C09104=1059.503,108.760,421.956,171.884,30.619,155.688
C09105=1059.497,108.511,421.976,171.883,30.616,155.687
C09106=1059.490,108.261,421.996,171.881,30.614,155.687
C09107=1059.484,108.012,422.014,171.879,30.611,155.687
C09108=1059.478,107.763,422.034,171.878,30.609,155.686
C09109=1059.472,107.514,422.053,171.876,30.606,155.686
C09110=1059.466,107.264,422.073,171.875,30.603,155.685
C09111=1059.460,107.015,422.093,171.873,30.601,155.685
C09112=1059.455,106.766,422.112,171.871,30.598,155.685
C09113=1059.448,106.517,422.131,171.870,30.596,155.684
C09114=1059.442,106.268,422.150,171.868,30.593,155.684
C09115=1059.437,106.019,422.170,171.867,30.591,155.683
C09116=1059.431,105.769,422.189,171.865,30.588,155.683
C09117=1059.424,105.521,422.208,171.863,30.585,155.683
C09118=1059.419,105.271,422.228,171.862,30.583,155.682
C09119=1059.413,105.022,422.247,171.861,30.580,155.682
C09120=1059.407,104.773,422.267,171.859,30.577,155.681
C09121=1059.401,104.524,422.286,171.857,30.575,155.681
C09122=1059.395,104.274,422.305,171.855,30.573,155.681
C09123=1059.389,104.025,422.324,171.854,30.570,155.680
C09124=1059.383,103.776,422.344,171.853,30.567,155.680
C09125=1059.377,103.527,422.363,171.851,30.565,155.679
C09126=1059.371,103.278,422.382,171.849,30.562,155.679
C09127=1059.365,103.028,422.401,171.847,30.559,155.679
C09128=1059.359,102.779,422.421,171.846,30.557,155.678
C09129=1059.354,102.531,422.440,171.845,30.554,155.678
C09130=1059.348,102.281,422.459,171.843,30.551,155.677
C09131=1059.342,102.032,422.478,171.841,30.549,155.677
C09132=1059.336,101.783,422.497,171.840,30.547,155.677
C09133=1059.330,101.534,422.517,171.839,30.544,155.676
C09134=1059.325,101.284,422.536,171.837,30.541,155.676
C09135=1059.318,101.035,422.555,171.835,30.539,155.675
C09136=1059.313,100.786,422.574,171.833,30.536,155.675
C09137=1059.306,100.537,422.593,171.832,30.533,155.675
C09138=1059.300,100.287,422.612,171.831,30.531,155.674
C09139=1059.295,100.038,422.631,171.829,30.529,155.674
C09140=1059.288,99.789,422.650,171.827,30.526,155.674
C09141=1059.283,99.539,422.669,171.825,30.523,155.673
C09142=1059.276,99.291,422.688,171.824,30.521,155.673
C09143=1059.270,99.041,422.708,171.823,30.518,155.672
C09144=1059.264,98.792,422.726,171.821,30.516,155.672
C09145=1059.258,98.543,422.746,171.819,30.513,155.672
C09146=1059.252,98.294,422.764,171.818,30.511,155.671
C09147=1059.247,98.045,422.783,171.817,30.508,155.671
C09148=1059.240,97.796,422.802,171.815,30.505,155.670
C09149=1059.234,97.546,422.821,171.813,30.503,155.670
C09150=1059.228,97.297,422.840,171.811,30.501,155.670
C09151=1059.222,97.048,422.859,171.810,30.498,155.669
C09152=1059.216,96.799,422.878,171.809,30.495,155.669
C09153=1059.210,96.549,422.897,171.807,30.493,155.668
C09154=1059.204,96.300,422.915,171.805,30.491,155.668
C09155=1059.198,96.051,422.935,171.804,30.488,155.668
C09156=1059.192,95.802,422.953,171.802,30.485,155.667
C09157=1059.187,95.553,422.972,171.801,30.483,155.667
C09158=1059.180,95.304,422.991,171.799,30.480,155.666
C09159=1059.175,95.054,423.010,171.797,30.477,155.666
C09160=1059.168,94.805,423.029,171.796,30.475,155.666
C09161=1059.162,94.520,423.050,171.795,30.472,155.665
C09162=1059.155,94.235,423.072,171.793,30.469,155.665
C09163=1059.148,93.951,423.093,171.791,30.466,155.664
C09164=1059.142,93.666,423.115,171.789,30.463,155.664
C09165=1059.135,93.417,423.133,171.788,30.461,155.663
C09166=1059.129,93.168,423.153,171.786,30.458,155.663
C09167=1059.123,92.919,423.171,171.784,30.455,155.663
C09168=1059.118,92.669,423.190,171.782,30.453,155.662
C09169=1059.111,92.420,423.208,171.781,30.451,155.662
C09170=1059.106,92.171,423.227,171.780,30.448,155.662
C09171=1059.100,91.922,423.246,171.778,30.445,155.661
C09172=1059.094,91.672,423.265,171.776,30.442,155.661
C09173=1059.088,91.423,423.284,171.775,30.440,155.660
C09174=1059.083,91.174,423.302,171.774,30.437,155.660
C09175=1059.076,90.925,423.321,171.772,30.435,155.660
C09176=1059.071,90.675,423.340,171.770,30.432,155.659
C09177=1059.064,90.426,423.358,171.769,30.430,155.659
C09178=1059.058,90.177,423.377,171.767,30.427,155.658
C09179=1059.052,89.927,423.395,171.766,30.424,155.658
C09180=1059.046,89.679,423.413,171.764,30.422,155.658
C09181=1059.040,89.429,423.433,171.763,30.420,155.657
C09182=1059.034,89.180,423.451,171.761,30.417,155.657
C09183=1059.028,88.931,423.469,171.759,30.415,155.656
C09184=1059.021,88.681,423.488,171.758,30.412,155.656
C09185=1059.015,88.432,423.507,171.756,30.410,155.656
C09186=1059.010,88.183,423.525,171.755,30.407,155.655
C09187=1059.004,87.934,423.543,171.753,30.405,155.655
C09188=1058.997,87.685,423.562,171.752,30.402,155.655
C09189=1058.991,87.435,423.580,171.750,30.400,155.654
C09190=1058.985,87.185,423.599,171.749,30.397,155.654
C09191=1058.979,86.937,423.617,171.747,30.395,155.653
C09192=1058.973,86.687,423.635,171.745,30.392,155.653
C09193=1058.967,86.438,423.654,171.744,30.389,155.653
C09194=1058.961,86.189,423.673,171.743,30.387,155.652
C09195=1058.956,85.940,423.691,171.741,30.384,155.652
C09196=1058.949,85.691,423.709,171.739,30.382,155.652
C09197=1058.943,85.442,423.728,171.738,30.379,155.651
C09198=1058.937,85.192,423.746,171.737,30.377,155.651
C09199=1058.931,84.943,423.764,171.735,30.374,155.650
C09200=1058.926,84.693,423.783,171.733,30.372,155.650
C09201=1058.919,84.444,423.801,171.731,30.369,155.650
C09202=1058.913,84.195,423.820,171.731,30.367,155.649
C09203=1058.907,83.946,423.838,171.729,30.364,155.649
C09204=1058.901,83.697,423.856,171.727,30.361,155.648
C09205=1058.895,83.447,423.875,171.725,30.359,155.648
C09206=1058.890,83.198,423.893,171.725,30.357,155.648
C09207=1058.883,82.949,423.911,171.723,30.354,155.647
C09208=1058.877,82.700,423.930,171.721,30.351,155.647
C09209=1058.871,82.450,423.948,171.719,30.349,155.646
C09210=1058.865,82.201,423.966,171.719,30.347,155.646
C09211=1058.860,81.951,423.984,171.717,30.344,155.646
C09212=1058.853,81.702,424.003,171.715,30.341,155.645
C09213=1058.848,81.453,424.021,171.713,30.338,155.645
C09214=1058.841,81.204,424.039,171.712,30.336,155.644
C09215=1058.835,80.954,424.057,171.711,30.334,155.644
C09216=1058.829,80.706,424.076,171.709,30.331,155.644
C09217=1058.823,80.456,424.093,171.707,30.328,155.643
C09218=1058.818,80.207,424.113,171.706,30.326,155.643
C09219=1058.812,79.958,424.130,171.705,30.323,155.643
C09220=1058.806,79.708,424.148,171.703,30.321,155.642
C09221=1058.800,79.460,424.166,171.701,30.318,155.642
C09222=1058.794,79.210,424.184,171.700,30.316,155.641
C09223=1058.788,78.961,424.203,171.699,30.313,155.641
C09224=1058.782,78.712,424.221,171.697,30.310,155.641
C09225=1058.773,78.312,424.250,171.694,30.306,155.640
C09226=1058.763,77.912,424.279,171.692,30.302,155.639
C09227=1058.753,77.512,424.308,171.690,30.298,155.639
C09228=1058.743,77.114,424.336,171.687,30.294,155.638
C09229=1058.737,76.864,424.354,171.685,30.292,155.638
C09230=1058.731,76.615,424.373,171.684,30.289,155.637
C09231=1058.725,76.366,424.391,171.683,30.287,155.637
C09232=1058.719,76.116,424.409,171.681,30.284,155.637
C09233=1058.713,75.867,424.427,171.679,30.282,155.636
C09234=1058.707,75.618,424.445,171.678,30.279,155.636
C09235=1058.701,75.368,424.463,171.677,30.277,155.635
C09236=1058.696,75.119,424.480,171.675,30.275,155.635
C09237=1058.689,74.870,424.498,171.673,30.272,155.635
C09238=1058.682,74.620,424.516,171.672,30.269,155.634
C09239=1058.677,74.371,424.534,171.671,30.267,155.634
C09240=1058.671,74.122,424.552,171.669,30.265,155.634
C09241=1058.665,73.873,424.570,171.667,30.262,155.633
C09242=1058.659,73.623,424.588,171.665,30.259,155.633
C09243=1058.653,73.374,424.606,171.665,30.257,155.632
C09244=1058.647,73.125,424.623,171.663,30.254,155.632
C09245=1058.641,72.876,424.642,171.661,30.252,155.632
C09246=1058.635,72.627,424.659,171.660,30.249,155.631
C09247=1058.628,72.377,424.677,171.659,30.246,155.631
C09248=1058.623,72.128,424.695,171.657,30.244,155.631
C09249=1058.617,71.878,424.713,171.655,30.242,155.630
C09250=1058.611,71.629,424.730,171.654,30.239,155.630
C09251=1058.605,71.380,424.749,171.652,30.237,155.630
C09252=1058.599,71.130,424.767,171.651,30.234,155.629
C09253=1058.592,70.882,424.784,171.649,30.232,155.629
C09254=1058.586,70.632,424.802,171.648,30.229,155.628
C09255=1058.581,70.383,424.819,171.646,30.227,155.628
C09256=1058.575,70.133,424.837,171.645,30.224,155.628
C09257=1058.569,69.884,424.855,171.643,30.221,155.627
C09258=1058.563,69.634,424.873,171.642,30.219,155.627
C09259=1058.557,69.386,424.890,171.640,30.217,155.626
C09260=1058.551,69.136,424.908,171.639,30.214,155.626
C09261=1058.541,68.752,424.935,171.636,30.210,155.625
C09262=1058.532,68.368,424.962,171.634,30.207,155.625
C09263=1058.522,67.985,424.989,171.632,30.203,155.624
C09264=1058.513,67.601,425.016,171.629,30.198,155.624
C09265=1058.508,67.352,425.034,171.628,30.196,155.623
C09266=1058.501,67.102,425.051,171.626,30.194,155.623
C09267=1058.495,66.852,425.069,171.625,30.191,155.623
C09268=1058.489,66.603,425.087,171.623,30.189,155.622
C09269=1058.483,66.354,425.104,171.622,30.186,155.622
C09270=1058.477,66.105,425.122,171.620,30.184,155.622
C09271=1058.471,65.855,425.140,171.619,30.181,155.621
C09272=1058.465,65.606,425.157,171.617,30.179,155.621
C09273=1058.459,65.357,425.175,171.616,30.176,155.620
C09274=1058.453,65.108,425.192,171.614,30.174,155.620
C09275=1058.447,64.859,425.209,171.613,30.171,155.620
C09276=1058.441,64.609,425.227,171.612,30.169,155.619
C09277=1058.435,64.360,425.245,171.610,30.166,155.619
C09278=1058.429,64.110,425.261,171.608,30.164,155.619
C09279=1058.422,63.860,425.279,171.607,30.161,155.618
C09280=1058.416,63.612,425.296,171.606,30.159,155.618
C09281=1058.409,63.362,425.313,171.604,30.157,155.617
C09282=1058.404,63.113,425.331,171.602,30.154,155.617
C09283=1058.397,62.864,425.348,171.600,30.152,155.617
C09284=1058.391,62.615,425.366,171.599,30.149,155.616
C09285=1058.384,62.330,425.385,171.597,30.146,155.616
C09286=1058.377,62.044,425.406,171.595,30.144,155.616
C09287=1058.370,61.760,425.425,171.594,30.141,155.615
C09288=1058.363,61.475,425.444,171.592,30.138,155.615
C09289=1058.357,61.226,425.462,171.591,30.136,155.614
C09290=1058.350,60.976,425.478,171.589,30.133,155.614
C09291=1058.345,60.727,425.496,171.588,30.131,155.614
C09292=1058.338,60.478,425.513,171.587,30.129,155.613
C09293=1058.332,60.229,425.530,171.585,30.126,155.613
C09294=1058.326,59.979,425.548,171.583,30.124,155.613
C09295=1058.320,59.730,425.565,171.581,30.121,155.612
C09296=1058.314,59.480,425.582,171.581,30.119,155.612
C09297=1058.307,59.231,425.599,171.579,30.116,155.612
C09298=1058.301,58.981,425.616,171.577,30.114,155.611
C09299=1058.295,58.732,425.634,171.575,30.112,155.611
C09300=1058.289,58.484,425.651,171.575,30.109,155.610
C09301=1058.283,58.233,425.668,171.573,30.106,155.610
C09302=1058.277,57.985,425.685,171.571,30.104,155.610
C09303=1058.270,57.735,425.702,171.569,30.101,155.609
C09304=1058.265,57.485,425.719,171.569,30.099,155.609
C09305=1058.258,57.236,425.736,171.567,30.097,155.609
C09306=1058.253,56.987,425.754,171.565,30.094,155.608
C09307=1058.247,56.738,425.770,171.563,30.092,155.608
C09308=1058.240,56.488,425.787,171.562,30.089,155.608
C09309=1058.234,56.239,425.805,171.561,30.087,155.607
C09310=1058.228,55.990,425.821,171.559,30.084,155.607
C09311=1058.221,55.740,425.839,171.557,30.082,155.606
C09312=1058.216,55.491,425.856,171.556,30.080,155.606
C09313=1058.209,55.241,425.873,171.555,30.077,155.606
C09314=1058.203,54.993,425.890,171.553,30.075,155.605
C09315=1058.198,54.743,425.907,171.551,30.072,155.605
C09316=1058.191,54.493,425.924,171.550,30.070,155.605
C09317=1058.185,54.244,425.942,171.549,30.067,155.604
C09318=1058.180,53.995,425.958,171.547,30.065,155.604
C09319=1058.173,53.746,425.975,171.545,30.063,155.604
C09320=1058.167,53.496,425.992,171.544,30.060,155.603
C09321=1058.161,53.247,426.009,171.543,30.057,155.603
C09322=1058.155,52.997,426.026,171.541,30.055,155.603
C09323=1058.149,52.748,426.043,171.539,30.052,155.602
C09324=1058.143,52.499,426.059,171.538,30.050,155.602
C09325=1058.136,52.249,426.077,171.537,30.048,155.601
C09326=1058.131,52.000,426.094,171.535,30.045,155.601
C09327=1058.125,51.751,426.111,171.533,30.043,155.601
C09328=1058.118,51.501,426.127,171.532,30.040,155.600
C09329=1058.113,51.252,426.145,171.531,30.037,155.600
C09330=1058.107,51.003,426.161,171.529,30.035,155.600
C09331=1058.101,50.754,426.178,171.527,30.033,155.599
C09332=1058.094,50.504,426.195,171.526,30.030,155.599
C09333=1058.089,50.255,426.212,171.525,30.028,155.599
C09334=1058.083,50.005,426.228,171.523,30.025,155.598
C09335=1058.076,49.757,426.245,171.522,30.023,155.598
C09336=1058.070,49.506,426.263,171.520,30.020,155.597
C09337=1058.065,49.257,426.279,171.519,30.018,155.597
C09338=1058.058,49.008,426.296,171.517,30.016,155.597
C09339=1058.053,48.759,426.313,171.516,30.013,155.596
C09340=1058.046,48.509,426.330,171.514,30.010,155.596
C09341=1058.040,48.260,426.346,171.513,30.008,155.596
C09342=1058.035,48.010,426.363,171.511,30.005,155.595
C09343=1058.029,47.761,426.380,171.510,30.003,155.595
C09344=1058.022,47.511,426.397,171.508,30.001,155.595
C09345=1058.016,47.263,426.414,171.507,29.998,155.594
C09346=1058.011,47.013,426.431,171.505,29.995,155.594
C09347=1058.005,46.764,426.447,171.504,29.993,155.593
C09348=1057.999,46.515,426.464,171.502,29.991,155.593
C09349=1057.992,46.229,426.483,171.501,29.988,155.593
C09350=1057.985,45.943,426.502,171.499,29.985,155.592
C09351=1057.978,45.659,426.521,171.497,29.982,155.592
C09352=1057.971,45.373,426.541,171.495,29.979,155.591
C09353=1057.965,45.124,426.557,171.494,29.977,155.591
C09354=1057.959,44.875,426.574,171.492,29.974,155.591
C09355=1057.953,44.626,426.590,171.491,29.972,155.590
C09356=1057.948,44.376,426.607,171.489,29.969,155.590
C09357=1057.942,44.127,426.623,171.488,29.967,155.590
C09358=1057.935,43.877,426.641,171.487,29.964,155.589
C09359=1057.929,43.628,426.657,171.485,29.962,155.589
C09360=1057.924,43.378,426.674,171.483,29.959,155.588
C09361=1057.918,43.129,426.690,171.482,29.957,155.588
C09362=1057.912,42.880,426.706,171.481,29.954,155.588
C09363=1057.905,42.630,426.724,171.479,29.952,155.587
C09364=1057.899,42.381,426.740,171.477,29.950,155.587
C09365=1057.893,42.132,426.756,171.476,29.947,155.587
C09366=1057.887,41.882,426.772,171.475,29.945,155.586
C09367=1057.881,41.633,426.789,171.473,29.943,155.586
C09368=1057.875,41.384,426.806,171.471,29.940,155.586
C09369=1057.869,41.134,426.822,171.470,29.937,155.585
C09370=1057.863,40.885,426.838,171.468,29.935,155.585
C09371=1057.857,40.635,426.855,171.467,29.932,155.585
C09372=1057.851,40.386,426.871,171.465,29.930,155.584
C09373=1057.845,40.137,426.887,171.464,29.928,155.584
C09374=1057.839,39.887,426.903,171.462,29.925,155.584
C09375=1057.832,39.637,426.920,171.461,29.923,155.583
C09376=1057.826,39.389,426.937,171.459,29.921,155.583
C09377=1057.820,39.139,426.953,171.458,29.918,155.583
C09378=1057.814,38.890,426.970,171.456,29.916,155.582
C09379=1057.808,38.641,426.986,171.455,29.913,155.582
C09380=1057.802,38.391,427.002,171.453,29.911,155.581
C09381=1057.796,38.142,427.018,171.452,29.908,155.581
C09382=1057.790,37.893,427.035,171.450,29.906,155.581
C09383=1057.784,37.642,427.051,171.449,29.904,155.580
C09384=1057.778,37.393,427.067,171.447,29.901,155.580
C09385=1057.772,37.144,427.084,171.446,29.899,155.580
C09386=1057.766,36.894,427.100,171.444,29.897,155.579
C09387=1057.759,36.645,427.116,171.443,29.894,155.579
C09388=1057.753,36.396,427.132,171.441,29.892,155.579
C09389=1057.747,36.147,427.148,171.440,29.889,155.578
C09390=1057.741,35.897,427.165,171.438,29.887,155.578
C09391=1057.735,35.647,427.181,171.437,29.884,155.578
C09392=1057.728,35.398,427.197,171.435,29.882,155.577
C09393=1057.722,35.149,427.213,171.434,29.879,155.577
C09394=1057.716,34.900,427.229,171.432,29.877,155.577
C09395=1057.710,34.650,427.245,171.431,29.875,155.576
C09396=1057.704,34.401,427.262,171.429,29.873,155.576
C09397=1057.698,34.152,427.278,171.428,29.870,155.576
C09398=1057.692,33.902,427.293,171.426,29.868,155.575
C09399=1057.686,33.653,427.309,171.424,29.866,155.575
C09400=1057.680,33.402,427.326,171.423,29.863,155.575
C09401=1057.674,33.153,427.342,171.422,29.861,155.574
C09402=1057.667,32.904,427.358,171.420,29.858,155.574
C09403=1057.661,32.655,427.374,171.418,29.856,155.574
C09404=1057.655,32.405,427.390,171.417,29.853,155.573
C09405=1057.649,32.156,427.406,171.416,29.851,155.573
C09406=1057.643,31.906,427.422,171.414,29.849,155.573
C09407=1057.637,31.657,427.438,171.412,29.846,155.572
C09408=1057.631,31.408,427.454,171.411,29.844,155.572
C09409=1057.625,31.158,427.470,171.410,29.842,155.572
C09410=1057.619,30.909,427.486,171.408,29.839,155.571
C09411=1057.613,30.660,427.503,171.406,29.837,155.571
C09412=1057.606,30.410,427.518,171.405,29.835,155.571
C09413=1057.599,30.125,427.537,171.404,29.832,155.570
C09414=1057.593,29.840,427.555,171.402,29.829,155.570
C09415=1057.586,29.554,427.573,171.399,29.826,155.569
C09416=1057.579,29.270,427.590,171.398,29.823,155.569
C09417=1057.573,29.020,427.607,171.397,29.821,155.569
C09418=1057.567,28.771,427.623,171.395,29.819,155.568
C09419=1057.561,28.521,427.639,171.393,29.817,155.568
C09420=1057.555,28.272,427.654,171.392,29.814,155.568
C09421=1057.549,28.022,427.670,171.391,29.812,155.567
C09422=1057.542,27.773,427.686,171.389,29.810,155.567
C09423=1057.536,27.523,427.702,171.387,29.807,155.567
C09424=1057.530,27.274,427.718,171.386,29.805,155.566
C09425=1057.524,27.025,427.734,171.385,29.802,155.566
C09426=1057.518,26.775,427.749,171.383,29.800,155.566
C09427=1057.511,26.526,427.765,171.381,29.798,155.565
C09428=1057.505,26.277,427.781,171.380,29.795,155.565
C09429=1057.500,26.027,427.797,171.378,29.793,155.565
C09430=1057.493,25.778,427.812,171.377,29.791,155.564
C09431=1057.487,25.528,427.828,171.375,29.788,155.564
C09432=1057.481,25.279,427.843,171.374,29.786,155.564
C09433=1057.475,25.029,427.860,171.372,29.784,155.564
C09434=1057.468,24.780,427.875,171.370,29.781,155.563
C09435=1057.462,24.530,427.891,171.369,29.779,155.563
C09436=1057.456,24.281,427.907,171.368,29.776,155.562
C09437=1057.450,24.031,427.922,171.366,29.774,155.562
C09438=1057.444,23.782,427.938,171.364,29.772,155.562
C09439=1057.437,23.533,427.954,171.363,29.769,155.561
C09440=1057.432,23.283,427.970,171.362,29.767,155.561
C09441=1057.425,23.034,427.985,171.360,29.765,155.561
C09442=1057.419,22.784,428.001,171.358,29.762,155.560
C09443=1057.413,22.535,428.016,171.356,29.760,155.560
C09444=1057.407,22.285,428.032,171.356,29.758,155.560
C09445=1057.400,22.036,428.048,171.354,29.755,155.559
C09446=1057.395,21.786,428.063,171.352,29.753,155.559
C09447=1057.388,21.537,428.079,171.350,29.751,155.559
C09448=1057.382,21.287,428.094,171.350,29.749,155.559
C09449=1057.376,21.039,428.110,171.348,29.746,155.558
C09450=1057.371,20.789,428.125,171.346,29.744,155.558
C09451=1057.364,20.540,428.141,171.344,29.741,155.558
C09452=1057.358,20.290,428.156,171.343,29.739,155.557
C09453=1057.352,20.041,428.172,171.342,29.737,155.557
C09454=1057.346,19.791,428.188,171.340,29.735,155.557
C09455=1057.339,19.542,428.203,171.338,29.732,155.556
C09456=1057.334,19.292,428.219,171.337,29.730,155.556
C09457=1057.327,19.042,428.234,171.335,29.727,155.556
C09458=1057.321,18.793,428.249,171.334,29.725,155.555
C09459=1057.316,18.544,428.265,171.332,29.723,155.555
C09460=1057.309,18.295,428.280,171.331,29.721,155.555
C09461=1057.303,18.045,428.296,171.329,29.718,155.554
C09462=1057.297,17.795,428.311,171.327,29.716,155.554
C09463=1057.290,17.546,428.326,171.326,29.714,155.554
C09464=1057.285,17.296,428.342,171.325,29.711,155.553
C09465=1057.278,17.047,428.358,171.323,29.709,155.553
C09466=1057.272,16.797,428.373,171.321,29.707,155.553
C09467=1057.266,16.548,428.388,171.319,29.704,155.552
C09468=1057.260,16.299,428.403,171.319,29.702,155.552
C09469=1057.254,16.049,428.419,171.317,29.700,155.552
C09470=1057.248,15.799,428.434,171.315,29.697,155.551
C09471=1057.241,15.550,428.450,171.313,29.695,155.551
C09472=1057.235,15.300,428.465,171.312,29.693,155.551
C09473=1057.230,15.051,428.480,171.311,29.691,155.551
C09474=1057.223,14.802,428.495,171.309,29.688,155.550
C09475=1057.217,14.552,428.511,171.307,29.686,155.550
C09476=1057.211,14.303,428.526,171.306,29.684,155.550
C09477=1057.204,14.020,428.543,171.304,29.681,155.549
C09478=1057.197,13.735,428.560,171.302,29.679,155.549
C09479=1057.190,13.451,428.577,171.301,29.676,155.549
C09480=1057.183,13.168,428.595,171.299,29.674,155.548
C09481=1057.177,12.918,428.610,171.297,29.671,155.548
C09482=1057.170,12.668,428.625,171.295,29.669,155.548
C09483=1057.164,12.419,428.640,171.295,29.667,155.547
C09484=1057.157,12.170,428.656,171.293,29.665,155.547
C09485=1057.151,11.921,428.670,171.291,29.663,155.547
C09486=1057.145,11.671,428.685,171.289,29.660,155.546
C09487=1057.139,11.421,428.701,171.288,29.658,155.546
C09488=1057.133,11.171,428.716,171.286,29.656,155.546
C09489=1057.127,10.922,428.731,171.285,29.654,155.546
C09490=1057.120,10.673,428.746,171.283,29.652,155.545
C09491=1057.114,10.424,428.761,171.282,29.649,155.545
C09492=1057.108,10.174,428.776,171.280,29.647,155.545
C09493=1057.101,9.925,428.791,171.278,29.644,155.544
C09494=1057.095,9.675,428.806,171.277,29.642,155.544
C09495=1057.089,9.425,428.821,171.276,29.640,155.544
C09496=1057.084,9.176,428.836,171.274,29.638,155.543
C09497=1057.077,8.926,428.851,171.272,29.636,155.543
C09498=1057.071,8.677,428.866,171.270,29.634,155.543
C09499=1057.064,8.428,428.881,171.269,29.631,155.543
C09500=1057.058,8.179,428.896,171.268,29.629,155.542
C09501=1057.052,7.929,428.911,171.266,29.627,155.542
C09502=1057.046,7.679,428.926,171.264,29.625,155.542
C09503=1057.039,7.430,428.941,171.263,29.622,155.541
C09504=1057.033,7.181,428.955,171.261,29.620,155.541
C09505=1057.028,6.931,428.971,171.260,29.618,155.541
C09506=1057.021,6.681,428.986,171.258,29.616,155.540
C09507=1057.015,6.431,429.001,171.257,29.613,155.540
C09508=1057.009,6.182,429.015,171.255,29.611,155.540
C09509=1057.003,5.933,429.030,171.253,29.609,155.540
C09510=1056.996,5.683,429.045,171.251,29.607,155.539
C09511=1056.991,5.434,429.060,171.251,29.605,155.539
C09512=1056.984,5.185,429.075,171.249,29.603,155.539
C09513=1056.978,4.935,429.090,171.247,29.600,155.538
C09514=1056.972,4.686,429.104,171.245,29.598,155.538
C09515=1056.966,4.436,429.119,171.244,29.596,155.538
C09516=1056.959,4.187,429.134,171.242,29.593,155.538
C09517=1056.953,3.937,429.149,171.241,29.591,155.537
C09518=1056.948,3.688,429.164,171.239,29.589,155.537
C09519=1056.942,3.437,429.179,171.238,29.587,155.537
C09520=1056.935,3.188,429.194,171.236,29.584,155.536
C09521=1056.930,2.939,429.208,171.234,29.582,155.536
C09522=1056.923,2.689,429.223,171.232,29.580,155.536
C09523=1056.917,2.439,429.238,171.232,29.578,155.535
C09524=1056.911,2.191,429.253,171.230,29.576,155.535
C09525=1056.905,1.941,429.268,171.228,29.574,155.535
C09526=1056.899,1.692,429.282,171.226,29.571,155.535
C09527=1056.893,1.442,429.297,171.225,29.569,155.534
C09528=1056.886,1.192,429.311,171.223,29.566,155.534
C09529=1056.881,0.943,429.326,171.222,29.564,155.534
C09530=1056.874,0.693,429.341,171.220,29.562,155.533
C09531=1056.868,0.444,429.356,171.219,29.560,155.533
C09532=1056.862,0.195,429.370,171.217,29.558,155.533
C09533=1056.856,-0.055,429.385,171.215,29.556,155.533
C09534=1056.850,-0.304,429.399,171.213,29.553,155.532
C09535=1056.844,-0.554,429.414,171.213,29.551,155.532
C09536=1056.838,-0.803,429.429,171.211,29.549,155.532
C09537=1056.832,-1.053,429.444,171.209,29.547,155.531
C09538=1056.825,-1.302,429.459,171.208,29.544,155.531
C09539=1056.820,-1.552,429.472,171.206,29.542,155.531
C09540=1056.814,-1.802,429.487,171.204,29.540,155.530
C09541=1056.807,-2.084,429.504,171.202,29.537,155.530
C09542=1056.801,-2.365,429.520,171.201,29.535,155.530
C09543=1056.794,-2.647,429.537,171.199,29.532,155.529
C09544=1056.786,-2.929,429.553,171.197,29.530,155.529
C09545=1056.780,-3.178,429.568,171.195,29.528,155.529
C09546=1056.774,-3.428,429.582,171.194,29.526,155.529
C09547=1056.768,-3.678,429.597,171.192,29.523,155.528
C09548=1056.762,-3.927,429.612,171.191,29.521,155.528
C09549=1056.756,-4.177,429.626,171.189,29.519,155.528
C09550=1056.750,-4.426,429.640,171.188,29.517,155.527
C09551=1056.743,-4.676,429.655,171.186,29.515,155.527
C09552=1056.737,-4.926,429.669,171.184,29.513,155.527
C09553=1056.731,-5.174,429.683,171.182,29.511,155.527
C09554=1056.724,-5.424,429.698,171.181,29.508,155.526
C09555=1056.719,-5.674,429.712,171.180,29.506,155.526
C09556=1056.712,-5.923,429.727,171.178,29.504,155.526
C09557=1056.706,-6.173,429.740,171.176,29.502,155.526
C09558=1056.700,-6.422,429.755,171.175,29.500,155.525
C09559=1056.693,-6.672,429.770,171.173,29.498,155.525
C09560=1056.687,-6.921,429.783,171.171,29.496,155.525
C09561=1056.681,-7.171,429.798,171.169,29.494,155.525
C09562=1056.675,-7.420,429.812,171.168,29.492,155.524
C09563=1056.669,-7.670,429.827,171.167,29.490,155.524
C09564=1056.663,-7.919,429.840,171.165,29.487,155.524
C09565=1056.656,-8.169,429.855,171.163,29.485,155.523
C09566=1056.651,-8.418,429.870,171.162,29.483,155.523
C09567=1056.644,-8.668,429.883,171.160,29.481,155.523
C09568=1056.638,-8.917,429.898,171.158,29.479,155.523
C09569=1056.632,-9.167,429.912,171.156,29.477,155.522
C09570=1056.625,-9.417,429.926,171.155,29.474,155.522
C09571=1056.619,-9.666,429.940,171.154,29.472,155.522
C09572=1056.614,-9.915,429.955,171.152,29.470,155.521
C09573=1056.607,-10.165,429.969,171.150,29.469,155.521
C09574=1056.601,-10.414,429.983,171.149,29.466,155.521
C09575=1056.595,-10.664,429.997,171.147,29.464,155.521
C09576=1056.589,-10.914,430.011,171.145,29.462,155.520
C09577=1056.582,-11.163,430.026,171.143,29.460,155.520
C09578=1056.577,-11.413,430.039,171.142,29.458,155.520
C09579=1056.570,-11.662,430.054,171.141,29.456,155.520
C09580=1056.564,-11.912,430.068,171.139,29.453,155.519
C09581=1056.558,-12.161,430.083,171.137,29.451,155.519
C09582=1056.552,-12.411,430.096,171.136,29.449,155.519
C09583=1056.545,-12.661,430.110,171.134,29.447,155.519
C09584=1056.540,-12.910,430.125,171.132,29.445,155.518
C09585=1056.533,-13.159,430.138,171.130,29.443,155.518
C09586=1056.527,-13.409,430.153,171.129,29.441,155.518
C09587=1056.522,-13.658,430.167,171.127,29.439,155.518
C09588=1056.515,-13.908,430.180,171.126,29.437,155.517
C09589=1056.509,-14.157,430.195,171.124,29.434,155.517
C09590=1056.503,-14.408,430.209,171.123,29.432,155.517
C09591=1056.497,-14.657,430.222,171.121,29.430,155.516
C09592=1056.491,-14.906,430.237,171.119,29.429,155.516
C09593=1056.485,-15.156,430.251,171.117,29.426,155.516
C09594=1056.479,-15.405,430.265,171.116,29.424,155.516
C09595=1056.472,-15.655,430.279,171.114,29.422,155.515
C09596=1056.466,-15.904,430.293,171.112,29.420,155.515
C09597=1056.459,-16.154,430.306,171.111,29.418,155.515
C09598=1056.454,-16.404,430.320,171.110,29.416,155.515
C09599=1056.447,-16.652,430.334,171.108,29.414,155.514
C09600=1056.441,-16.903,430.348,171.106,29.412,155.514
C09601=1056.435,-17.152,430.362,171.104,29.410,155.514
C09602=1056.428,-17.402,430.375,171.103,29.408,155.514
C09603=1056.422,-17.651,430.390,171.101,29.406,155.514
C09604=1056.416,-17.900,430.403,171.099,29.404,155.513
C09605=1056.409,-18.181,430.419,171.098,29.401,155.513
C09606=1056.402,-18.461,430.434,171.096,29.399,155.513
C09607=1056.395,-18.742,430.450,171.094,29.397,155.512
C09608=1056.389,-19.022,430.466,171.092,29.395,155.512
C09609=1056.382,-19.271,430.479,171.091,29.393,155.512
C09610=1056.376,-19.521,430.492,171.089,29.391,155.512
C09611=1056.370,-19.770,430.507,171.087,29.389,155.511
C09612=1056.364,-20.020,430.520,171.085,29.387,155.511
C09613=1056.358,-20.270,430.535,171.084,29.385,155.511
C09614=1056.351,-20.519,430.548,171.082,29.383,155.511
C09615=1056.345,-20.768,430.561,171.080,29.381,155.510
C09616=1056.339,-21.019,430.575,171.078,29.378,155.510
C09617=1056.333,-21.268,430.589,171.077,29.377,155.510
C09618=1056.326,-21.517,430.603,171.075,29.375,155.510
C09619=1056.320,-21.767,430.617,171.074,29.373,155.509
C09620=1056.314,-22.016,430.630,171.072,29.371,155.509
C09621=1056.308,-22.266,430.644,171.071,29.369,155.509
C09622=1056.302,-22.516,430.658,171.069,29.367,155.509
C09623=1056.295,-22.765,430.671,171.067,29.364,155.509
C09624=1056.290,-23.015,430.685,171.065,29.363,155.508
C09625=1056.283,-23.264,430.698,171.064,29.361,155.508
C09626=1056.277,-23.514,430.712,171.062,29.358,155.508
C09627=1056.271,-23.763,430.725,171.060,29.357,155.508
C09628=1056.265,-24.013,430.739,171.058,29.355,155.507
C09629=1056.259,-24.263,430.753,171.057,29.352,155.507
C09630=1056.253,-24.512,430.766,171.055,29.351,155.507
C09631=1056.247,-24.761,430.780,171.053,29.349,155.507
C09632=1056.241,-25.012,430.794,171.052,29.347,155.506
C09633=1056.234,-25.261,430.807,171.050,29.345,155.506
C09634=1056.228,-25.510,430.820,171.049,29.343,155.506
C09635=1056.223,-25.760,430.834,171.047,29.341,155.506
C09636=1056.216,-26.010,430.848,171.045,29.339,155.506
C09637=1056.210,-26.259,430.861,171.043,29.337,155.505
C09638=1056.204,-26.509,430.875,171.042,29.335,155.505
C09639=1056.198,-26.758,430.888,171.040,29.332,155.505
C09640=1056.191,-27.008,430.902,171.038,29.331,155.505
C09641=1056.185,-27.257,430.915,171.036,29.329,155.504
C09642=1056.179,-27.506,430.928,171.035,29.327,155.504
C09643=1056.174,-27.757,430.942,171.033,29.325,155.504
C09644=1056.167,-28.006,430.955,171.031,29.323,155.504
C09645=1056.161,-28.256,430.968,171.029,29.321,155.503
C09646=1056.154,-28.505,430.982,171.028,29.319,155.503
C09647=1056.148,-28.754,430.995,171.027,29.317,155.503
C09648=1056.141,-29.004,431.009,171.025,29.316,155.503
C09649=1056.135,-29.254,431.022,171.023,29.314,155.503
C09650=1056.129,-29.503,431.034,171.022,29.312,155.502
C09651=1056.124,-29.753,431.048,171.020,29.310,155.502
C09652=1056.117,-30.003,431.062,171.018,29.308,155.502
C09653=1056.111,-30.252,431.075,171.016,29.306,155.502
C09654=1056.105,-30.501,431.088,171.015,29.304,155.502
C09655=1056.098,-30.751,431.102,171.013,29.302,155.501
C09656=1056.092,-31.001,431.115,171.011,29.301,155.501
C09657=1056.086,-31.251,431.128,171.009,29.298,155.501
C09658=1056.079,-31.500,431.141,171.008,29.297,155.501
C09659=1056.073,-31.749,431.154,171.006,29.295,155.500
C09660=1056.067,-31.999,431.167,171.004,29.293,155.500
C09661=1056.061,-32.249,431.181,171.002,29.291,155.500
C09662=1056.055,-32.499,431.195,171.000,29.289,155.500
C09663=1056.049,-32.748,431.208,170.999,29.287,155.500
C09664=1056.043,-32.998,431.220,170.997,29.285,155.499
C09665=1056.037,-33.247,431.234,170.995,29.283,155.499
C09666=1056.030,-33.496,431.247,170.993,29.281,155.499
C09667=1056.024,-33.746,431.261,170.992,29.279,155.499
C09668=1056.018,-33.996,431.273,170.990,29.278,155.499
C09669=1056.011,-34.275,431.287,170.988,29.275,155.498
C09670=1056.004,-34.555,431.303,170.986,29.273,155.498
C09671=1055.997,-34.834,431.317,170.985,29.272,155.498
C09672=1055.990,-35.114,431.332,170.983,29.269,155.498
C09673=1055.984,-35.364,431.345,170.981,29.267,155.497
C09674=1055.978,-35.613,431.358,170.979,29.266,155.497
C09675=1055.972,-35.863,431.371,170.978,29.263,155.497
C09676=1055.966,-36.112,431.385,170.976,29.262,155.497
C09677=1055.960,-36.362,431.397,170.974,29.260,155.497
C09678=1055.954,-36.611,431.410,170.972,29.258,155.496
C09679=1055.947,-36.860,431.424,170.971,29.256,155.496
C09680=1055.942,-37.110,431.436,170.969,29.254,155.496
C09681=1055.935,-37.360,431.449,170.967,29.253,155.496
C09682=1055.929,-37.610,431.462,170.965,29.250,155.496
C09683=1055.923,-37.859,431.476,170.964,29.249,155.495
C09684=1055.917,-38.109,431.488,170.962,29.247,155.495
C09685=1055.910,-38.359,431.501,170.960,29.245,155.495
C09686=1055.904,-38.608,431.515,170.958,29.243,155.495
C09687=1055.898,-38.858,431.527,170.957,29.241,155.495
C09688=1055.892,-39.107,431.541,170.955,29.240,155.494
C09689=1055.886,-39.357,431.553,170.953,29.238,155.494
C09690=1055.880,-39.606,431.566,170.951,29.236,155.494
C09691=1055.874,-39.856,431.579,170.950,29.234,155.494
C09692=1055.867,-40.105,431.592,170.948,29.232,155.494
C09693=1055.861,-40.356,431.605,170.946,29.231,155.493
C09694=1055.855,-40.605,431.617,170.944,29.229,155.493
C09695=1055.849,-40.855,431.630,170.942,29.227,155.493
C09696=1055.843,-41.105,431.643,170.941,29.225,155.493
C09697=1055.836,-41.354,431.656,170.939,29.224,155.493
C09698=1055.830,-41.603,431.668,170.937,29.222,155.493
C09699=1055.824,-41.853,431.681,170.935,29.220,155.492
C09700=1055.818,-42.103,431.694,170.934,29.218,155.492
C09701=1055.811,-42.352,431.707,170.932,29.217,155.492
C09702=1055.805,-42.601,431.719,170.930,29.215,155.492
C09703=1055.799,-42.851,431.732,170.928,29.213,155.492
C09704=1055.793,-43.101,431.745,170.926,29.211,155.491
C09705=1055.787,-43.350,431.758,170.925,29.210,155.491
C09706=1055.781,-43.600,431.771,170.923,29.208,155.491
C09707=1055.774,-43.849,431.783,170.921,29.206,155.491
C09708=1055.768,-44.099,431.795,170.919,29.204,155.491
C09709=1055.762,-44.348,431.809,170.918,29.203,155.491
C09710=1055.756,-44.598,431.821,170.916,29.200,155.490
C09711=1055.750,-44.848,431.834,170.914,29.199,155.490
C09712=1055.743,-45.097,431.846,170.912,29.197,155.490
C09713=1055.737,-45.347,431.859,170.911,29.196,155.490
C09714=1055.731,-45.597,431.871,170.909,29.194,155.490
C09715=1055.725,-45.846,431.885,170.907,29.192,155.489
C09716=1055.718,-46.096,431.897,170.905,29.190,155.489
C09717=1055.712,-46.346,431.909,170.903,29.189,155.489
C09718=1055.706,-46.595,431.922,170.902,29.187,155.489
C09719=1055.700,-46.845,431.935,170.900,29.185,155.489
C09720=1055.694,-47.094,431.947,170.898,29.183,155.489
C09721=1055.688,-47.344,431.960,170.896,29.182,155.488
C09722=1055.682,-47.594,431.972,170.895,29.180,155.488
C09723=1055.676,-47.843,431.985,170.893,29.178,155.488
C09724=1055.669,-48.093,431.997,170.891,29.177,155.488
C09725=1055.663,-48.343,432.010,170.889,29.174,155.488
C09726=1055.657,-48.593,432.023,170.888,29.173,155.488
C09727=1055.652,-48.841,432.035,170.886,29.171,155.487
C09728=1055.645,-49.091,432.047,170.884,29.170,155.487
C09729=1055.639,-49.341,432.060,170.882,29.168,155.487
C09730=1055.633,-49.591,432.072,170.880,29.166,155.487
C09731=1055.627,-49.840,432.085,170.879,29.164,155.487
C09732=1055.620,-50.089,432.098,170.877,29.163,155.487
C09733=1055.614,-50.369,432.111,170.875,29.161,155.486
C09734=1055.607,-50.650,432.125,170.873,29.159,155.486
C09735=1055.599,-50.930,432.140,170.871,29.157,155.486
C09736=1055.593,-51.210,432.153,170.869,29.155,155.486
C09737=1055.586,-51.459,432.165,170.867,29.154,155.486
C09738=1055.580,-51.709,432.177,170.865,29.152,155.486
C09739=1055.573,-51.959,432.189,170.864,29.150,155.485
C09740=1055.567,-52.208,432.202,170.862,29.149,155.485
C09741=1055.561,-52.457,432.214,170.860,29.148,155.485
C09742=1055.555,-52.707,432.227,170.858,29.146,155.485
C09743=1055.548,-52.957,432.239,170.856,29.145,155.485
C09744=1055.541,-53.206,432.251,170.855,29.143,155.485
C09745=1055.535,-53.456,432.263,170.853,29.141,155.485
C09746=1055.529,-53.706,432.275,170.851,29.140,155.484
C09747=1055.523,-53.955,432.288,170.849,29.138,155.484
C09748=1055.517,-54.205,432.300,170.847,29.137,155.484
C09749=1055.510,-54.454,432.312,170.846,29.135,155.484
C09750=1055.504,-54.704,432.324,170.844,29.133,155.484
C09751=1055.498,-54.954,432.336,170.842,29.132,155.484
C09752=1055.492,-55.204,432.349,170.840,29.131,155.484
C09753=1055.485,-55.453,432.361,170.838,29.129,155.483
C09754=1055.478,-55.703,432.373,170.837,29.127,155.483
C09755=1055.472,-55.953,432.385,170.834,29.126,155.483
C09756=1055.466,-56.201,432.397,170.832,29.124,155.483
C09757=1055.461,-56.451,432.409,170.830,29.122,155.483
C09758=1055.454,-56.701,432.421,170.829,29.121,155.483
C09759=1055.448,-56.951,432.432,170.827,29.119,155.483
C09760=1055.442,-57.201,432.445,170.825,29.118,155.483
C09761=1055.435,-57.451,432.457,170.823,29.116,155.482
C09762=1055.429,-57.699,432.469,170.821,29.115,155.482
C09763=1055.423,-57.949,432.481,170.820,29.113,155.482
C09764=1055.416,-58.199,432.493,170.818,29.112,155.482
C09765=1055.410,-58.449,432.506,170.816,29.110,155.482
C09766=1055.404,-58.698,432.518,170.814,29.108,155.482
C09767=1055.397,-58.948,432.530,170.812,29.107,155.482
C09768=1055.392,-59.198,432.541,170.811,29.106,155.481
C09769=1055.386,-59.447,432.553,170.809,29.104,155.481
C09770=1055.379,-59.697,432.565,170.807,29.103,155.481
C09771=1055.373,-59.947,432.577,170.805,29.101,155.481
C09772=1055.366,-60.196,432.589,170.803,29.099,155.481
C09773=1055.360,-60.445,432.601,170.802,29.098,155.481
C09774=1055.355,-60.696,432.613,170.800,29.097,155.481
C09775=1055.348,-60.945,432.625,170.798,29.095,155.481
C09776=1055.341,-61.195,432.637,170.796,29.093,155.480
C09777=1055.336,-61.444,432.649,170.794,29.092,155.480
C09778=1055.329,-61.694,432.661,170.792,29.091,155.480
C09779=1055.323,-61.944,432.672,170.790,29.089,155.480
C09780=1055.317,-62.194,432.685,170.788,29.087,155.480
C09781=1055.311,-62.443,432.696,170.786,29.086,155.480
C09782=1055.305,-62.692,432.708,170.785,29.084,155.480
C09783=1055.299,-62.943,432.720,170.783,29.083,155.480
C09784=1055.293,-63.191,432.732,170.781,29.081,155.479
C09785=1055.286,-63.441,432.744,170.779,29.080,155.479
C09786=1055.280,-63.691,432.756,170.777,29.078,155.479
C09787=1055.274,-63.941,432.767,170.776,29.077,155.479
C09788=1055.268,-64.190,432.779,170.774,29.076,155.479
C09789=1055.262,-64.440,432.792,170.772,29.074,155.479
C09790=1055.256,-64.690,432.803,170.770,29.072,155.479
C09791=1055.250,-64.939,432.814,170.768,29.071,155.479
C09792=1055.243,-65.189,432.826,170.767,29.070,155.478
C09793=1055.237,-65.439,432.838,170.765,29.068,155.478
C09794=1055.231,-65.688,432.850,170.762,29.066,155.478
C09795=1055.225,-65.937,432.862,170.760,29.065,155.478
C09796=1055.219,-66.188,432.874,170.758,29.064,155.478
C09797=1055.212,-66.469,432.886,170.757,29.062,155.478
C09798=1055.205,-66.750,432.900,170.755,29.060,155.478
C09799=1055.198,-67.031,432.913,170.752,29.058,155.478
C09800=1055.191,-67.312,432.927,170.750,29.057,155.477
C09801=1055.185,-67.562,432.938,170.749,29.055,155.477
C09802=1055.179,-67.812,432.950,170.747,29.054,155.477
C09803=1055.174,-68.062,432.961,170.745,29.053,155.477
C09804=1055.167,-68.311,432.973,170.743,29.051,155.477
C09805=1055.161,-68.560,432.985,170.741,29.050,155.477
C09806=1055.154,-68.810,432.996,170.740,29.048,155.477
C09807=1055.149,-69.060,433.009,170.738,29.047,155.477
C09808=1055.143,-69.310,433.019,170.736,29.046,155.477
C09809=1055.136,-69.559,433.031,170.733,29.044,155.476
C09810=1055.130,-69.809,433.042,170.731,29.042,155.476
C09811=1055.125,-70.059,433.055,170.730,29.041,155.476
C09812=1055.118,-70.309,433.066,170.728,29.040,155.476
C09813=1055.112,-70.558,433.078,170.726,29.038,155.476
C09814=1055.106,-70.808,433.089,170.724,29.037,155.476
C09815=1055.100,-71.057,433.101,170.722,29.035,155.476
C09816=1055.094,-71.307,433.112,170.721,29.034,155.476
C09817=1055.088,-71.556,433.124,170.719,29.033,155.476
C09818=1055.082,-71.806,433.135,170.717,29.031,155.475
C09819=1055.076,-72.055,433.147,170.715,29.029,155.475
C09820=1055.070,-72.306,433.159,170.713,29.028,155.475
C09821=1055.064,-72.556,433.170,170.712,29.027,155.475
C09822=1055.058,-72.805,433.181,170.710,29.026,155.475
C09823=1055.051,-73.055,433.193,170.707,29.024,155.475
C09824=1055.046,-73.304,433.205,170.705,29.022,155.475
C09825=1055.040,-73.554,433.216,170.703,29.021,155.475
C09826=1055.034,-73.804,433.227,170.702,29.020,155.475
C09827=1055.027,-74.053,433.239,170.700,29.019,155.475
C09828=1055.022,-74.303,433.250,170.698,29.017,155.474
C09829=1055.015,-74.552,433.262,170.696,29.016,155.474
C09830=1055.009,-74.802,433.273,170.694,29.014,155.474
C09831=1055.003,-75.052,433.284,170.693,29.013,155.474
C09832=1054.997,-75.301,433.296,170.691,29.012,155.474
C09833=1054.991,-75.551,433.307,170.689,29.011,155.474
C09834=1054.984,-75.801,433.318,170.687,29.010,155.474
C09835=1054.978,-76.050,433.330,170.684,29.008,155.474
C09836=1054.972,-76.300,433.341,170.682,29.007,155.474
C09837=1054.966,-76.550,433.352,170.681,29.005,155.474
C09838=1054.960,-76.800,433.363,170.679,29.004,155.474
C09839=1054.954,-77.049,433.375,170.677,29.003,155.474
C09840=1054.947,-77.299,433.386,170.675,29.001,155.474
C09841=1054.942,-77.549,433.397,170.673,29.000,155.474
C09842=1054.935,-77.799,433.408,170.672,28.999,155.473
C09843=1054.929,-78.048,433.419,170.670,28.998,155.473
C09844=1054.923,-78.298,433.431,170.668,28.997,155.473
C09845=1054.917,-78.547,433.442,170.666,28.995,155.473
C09846=1054.911,-78.798,433.453,170.663,28.994,155.473
C09847=1054.905,-79.046,433.464,170.662,28.993,155.473
C09848=1054.899,-79.296,433.475,170.660,28.991,155.473
C09849=1054.892,-79.546,433.486,170.658,28.990,155.473
C09850=1054.886,-79.795,433.497,170.656,28.989,155.473
C09851=1054.880,-80.045,433.508,170.654,28.988,155.473
C09852=1054.874,-80.295,433.519,170.652,28.987,155.473
C09853=1054.867,-80.545,433.531,170.651,28.986,155.473
C09854=1054.861,-80.794,433.541,170.649,28.985,155.473
C09855=1054.855,-81.044,433.552,170.646,28.983,155.473
C09856=1054.849,-81.293,433.563,170.644,28.982,155.472
C09857=1054.843,-81.544,433.575,170.642,28.981,155.472
C09858=1054.836,-81.793,433.585,170.640,28.980,155.472
C09859=1054.830,-82.043,433.596,170.639,28.979,155.472
C09860=1054.824,-82.292,433.607,170.637,28.978,155.472
C09861=1054.816,-82.576,433.620,170.635,28.976,155.472
C09862=1054.809,-82.859,433.632,170.632,28.975,155.472
C09863=1054.802,-83.143,433.645,170.630,28.974,155.472
C09864=1054.795,-83.427,433.657,170.628,28.972,155.472
C09865=1054.789,-83.676,433.668,170.626,28.971,155.472
C09866=1054.783,-83.926,433.678,170.624,28.970,155.472
C09867=1054.776,-84.175,433.689,170.622,28.969,155.472
C09868=1054.770,-84.425,433.700,170.620,28.968,155.472
C09869=1054.764,-84.675,433.711,170.618,28.967,155.472
C09870=1054.758,-84.925,433.722,170.617,28.966,155.472
C09871=1054.751,-85.174,433.733,170.614,28.964,155.472
C09872=1054.745,-85.424,433.744,170.612,28.963,155.472
C09873=1054.740,-85.673,433.755,170.610,28.962,155.472
C09874=1054.733,-85.923,433.765,170.608,28.961,155.472
C09875=1054.727,-86.173,433.776,170.606,28.960,155.472
C09876=1054.721,-86.423,433.787,170.605,28.959,155.472
C09877=1054.714,-86.672,433.798,170.603,28.958,155.472
C09878=1054.708,-86.922,433.808,170.601,28.957,155.472
C09879=1054.702,-87.172,433.820,170.599,28.956,155.471
C09880=1054.696,-87.421,433.830,170.596,28.954,155.471
C09881=1054.690,-87.671,433.841,170.594,28.953,155.471
C09882=1054.683,-87.921,433.852,170.593,28.952,155.471
C09883=1054.677,-88.170,433.862,170.591,28.951,155.471
C09884=1054.671,-88.419,433.873,170.589,28.950,155.471
C09885=1054.665,-88.670,433.885,170.587,28.949,155.471
C09886=1054.659,-88.919,433.894,170.585,28.948,155.471
C09887=1054.653,-89.169,433.905,170.583,28.947,155.471
C09888=1054.647,-89.419,433.916,170.581,28.945,155.471
C09889=1054.640,-89.668,433.927,170.579,28.944,155.471
C09890=1054.634,-89.918,433.937,170.577,28.943,155.471
C09891=1054.628,-90.168,433.949,170.575,28.942,155.471
C09892=1054.622,-90.417,433.959,170.573,28.941,155.471
C09893=1054.616,-90.667,433.969,170.571,28.940,155.471
C09894=1054.610,-90.917,433.980,170.570,28.939,155.471
C09895=1054.603,-91.167,433.991,170.568,28.938,155.471
C09896=1054.598,-91.416,434.001,170.565,28.937,155.471
C09897=1054.591,-91.665,434.012,170.563,28.936,155.471
C09898=1054.585,-91.916,434.022,170.561,28.935,155.471
C09899=1054.579,-92.166,434.033,170.559,28.934,155.471
C09900=1054.573,-92.415,434.043,170.558,28.933,155.471
C09901=1054.567,-92.664,434.054,170.556,28.932,155.471
C09902=1054.561,-92.914,434.066,170.554,28.931,155.471
C09903=1054.555,-93.164,434.075,170.552,28.930,155.471
C09904=1054.549,-93.414,434.086,170.549,28.929,155.471
C09905=1054.542,-93.663,434.096,170.547,28.928,155.471
C09906=1054.536,-93.913,434.108,170.546,28.926,155.471
C09907=1054.531,-94.163,434.118,170.544,28.925,155.471
C09908=1054.524,-94.412,434.128,170.542,28.924,155.471
C09909=1054.518,-94.662,434.139,170.540,28.924,155.471
C09910=1054.512,-94.912,434.149,170.538,28.923,155.471
C09911=1054.506,-95.162,434.160,170.536,28.922,155.471
C09912=1054.500,-95.411,434.171,170.533,28.921,155.471
C09913=1054.494,-95.661,434.180,170.532,28.920,155.471
C09914=1054.488,-95.911,434.191,170.530,28.919,155.471
C09915=1054.481,-96.160,434.202,170.528,28.918,155.470
C09916=1054.476,-96.411,434.212,170.526,28.917,155.470
C09917=1054.470,-96.660,434.223,170.524,28.916,155.470
C09918=1054.464,-96.909,434.233,170.522,28.915,155.470
C09919=1054.458,-97.159,434.243,170.521,28.914,155.470
C09920=1054.452,-97.409,434.253,170.518,28.913,155.470
C09921=1054.446,-97.659,434.264,170.516,28.912,155.470
C09922=1054.439,-97.909,434.274,170.514,28.911,155.470
C09923=1054.433,-98.158,434.284,170.512,28.910,155.470
C09924=1054.427,-98.408,434.295,170.510,28.909,155.470
C09925=1054.420,-98.693,434.307,170.507,28.908,155.470
C09926=1054.413,-98.979,434.319,170.506,28.907,155.470
C09927=1054.406,-99.265,434.330,170.504,28.906,155.470
C09928=1054.399,-99.551,434.342,170.501,28.905,155.470
C09929=1054.392,-99.800,434.352,170.499,28.904,155.470
C09930=1054.386,-100.050,434.362,170.497,28.903,155.470
C09931=1054.380,-100.300,434.372,170.495,28.902,155.470
C09932=1054.374,-100.550,434.382,170.492,28.902,155.471
C09933=1054.367,-100.799,434.393,170.491,28.901,155.471
C09934=1054.362,-101.049,434.403,170.489,28.900,155.470
C09935=1054.355,-101.299,434.413,170.487,28.899,155.471
C09936=1054.349,-101.548,434.423,170.485,28.898,155.471
C09937=1054.343,-101.798,434.434,170.483,28.897,155.470
C09938=1054.337,-102.048,434.443,170.481,28.897,155.471
C09939=1054.330,-102.298,434.454,170.478,28.896,155.471
C09940=1054.325,-102.548,434.464,170.477,28.895,155.471
C09941=1054.318,-102.797,434.474,170.475,28.894,155.471
C09942=1054.312,-103.047,434.484,170.473,28.893,155.471
C09943=1054.307,-103.297,434.494,170.471,28.893,155.471
C09944=1054.300,-103.546,434.504,170.469,28.892,155.471
C09945=1054.294,-103.796,434.514,170.467,28.891,155.471
C09946=1054.287,-104.045,434.524,170.464,28.890,155.471
C09947=1054.282,-104.295,434.534,170.463,28.889,155.471
C09948=1054.275,-104.545,434.544,170.461,28.889,155.471
C09949=1054.269,-104.795,434.554,170.459,28.887,155.471
C09950=1054.263,-105.045,434.565,170.457,28.887,155.471
C09951=1054.257,-105.295,434.574,170.455,28.886,155.471
C09952=1054.251,-105.544,434.584,170.453,28.885,155.471
C09953=1054.245,-105.794,434.594,170.450,28.884,155.471
C09954=1054.239,-106.044,434.604,170.448,28.883,155.471
C09955=1054.233,-106.293,434.614,170.447,28.883,155.471
C09956=1054.226,-106.543,434.624,170.445,28.882,155.471
C09957=1054.220,-106.792,434.634,170.443,28.881,155.471
C09958=1054.215,-107.042,434.644,170.441,28.880,155.471
C09959=1054.208,-107.292,434.654,170.439,28.880,155.471
C09960=1054.202,-107.541,434.664,170.436,28.879,155.471
C09961=1054.196,-107.791,434.673,170.434,28.878,155.471
C09962=1054.189,-108.041,434.684,170.432,28.878,155.471
C09963=1054.184,-108.291,434.694,170.431,28.877,155.471
C09964=1054.177,-108.541,434.704,170.429,28.876,155.471
C09965=1054.171,-108.791,434.713,170.427,28.875,155.471
C09966=1054.165,-109.040,434.723,170.424,28.875,155.471
C09967=1054.159,-109.290,434.733,170.422,28.874,155.471
C09968=1054.152,-109.540,434.743,170.420,28.873,155.471
C09969=1054.146,-109.789,434.752,170.418,28.873,155.471
C09970=1054.140,-110.039,434.762,170.416,28.872,155.471
C09971=1054.134,-110.288,434.772,170.415,28.871,155.472
C09972=1054.128,-110.539,434.782,170.412,28.871,155.472
C09973=1054.122,-110.788,434.792,170.410,28.870,155.472
C09974=1054.116,-111.038,434.801,170.408,28.869,155.472
C09975=1054.110,-111.288,434.811,170.406,28.869,155.472
C09976=1054.103,-111.537,434.821,170.404,28.868,155.472
C09977=1054.097,-111.787,434.831,170.402,28.868,155.472
C09978=1054.091,-112.037,434.840,170.400,28.867,155.472
C09979=1054.085,-112.287,434.850,170.398,28.866,155.472
C09980=1054.078,-112.536,434.859,170.396,28.865,155.472
C09981=1054.072,-112.786,434.869,170.394,28.865,155.472
C09982=1054.067,-113.036,434.879,170.392,28.864,155.472
C09983=1054.061,-113.286,434.889,170.390,28.864,155.472
C09984=1054.054,-113.536,434.898,170.388,28.863,155.472
C09985=1054.048,-113.786,434.908,170.385,28.862,155.472
C09986=1054.042,-114.035,434.918,170.383,28.861,155.472
C09987=1054.036,-114.284,434.927,170.381,28.861,155.472
C09988=1054.030,-114.534,434.937,170.379,28.861,155.472
C09989=1054.023,-114.819,434.947,170.377,28.859,155.472
C09990=1054.015,-115.103,434.959,170.375,28.859,155.473
C09991=1054.009,-115.387,434.969,170.373,28.859,155.473
C09992=1054.001,-115.672,434.980,170.370,28.858,155.473
C09993=1053.995,-115.921,434.990,170.368,28.858,155.473
C09994=1053.990,-116.170,434.999,170.366,28.856,155.473
C09995=1053.984,-116.420,435.009,170.364,28.856,155.473
C09996=1053.977,-116.670,435.018,170.361,28.855,155.473
//INST
///DATE 2021/06/25 14:46
///ATTR SC,RW,RJ
////FRAME ROBOT
///GROUP1 RB1
NOP
MOVL C00000 V=800.0 PL=0
MOVL C00001 V=800.0 PL=0
MOVL C00002 V=800.0 PL=0
MOVL C00003 V=800.0 PL=0
MOVL C00004 V=800.0 PL=0
MOVL C00005 V=800.0 PL=0
MOVL C00006 V=800.0 PL=0
MOVL C00007 V=800.0 PL=0
MOVL C00008 V=800.0 PL=0
MOVL C00009 V=800.0 PL=0
MOVL C00010 V=800.0 PL=0
MOVL C00011 V=800.0 PL=0
MOVL C00012 V=800.0 PL=0
MOVL C00013 V=800.0 PL=0
MOVL C00014 V=800.0 PL=0
MOVL C00015 V=800.0 PL=0
MOVL C00016 V=800.0 PL=0
MOVL C00017 V=800.0 PL=0
MOVL C00018 V=800.0 PL=0
MOVL C00019 V=800.0 PL=0
MOVL C00020 V=800.0 PL=0
MOVL C00021 V=800.0 PL=0
MOVL C00022 V=800.0 PL=0
MOVL C00023 V=800.0 PL=0
MOVL C00024 V=800.0 PL=0
MOVL C00025 V=800.0 PL=0
MOVL C00026 V=800.0 PL=0
MOVL C00027 V=800.0 PL=0
MOVL C00028 V=800.0 PL=0
MOVL C00029 V=800.0 PL=0
MOVL C00030 V=800.0 PL=0
MOVL C00031 V=800.0 PL=0
MOVL C00032 V=800.0 PL=0
MOVL C00033 V=800.0 PL=0
MOVL C00034 V=800.0 PL=0
MOVL C00035 V=800.0 PL=0
MOVL C00036 V=800.0 PL=0
MOVL C00037 V=800.0 PL=0
MOVL C00038 V=800.0 PL=0
MOVL C00039 V=800.0 PL=0
MOVL C00040 V=800.0 PL=0
MOVL C00041 V=800.0 PL=0
MOVL C00042 V=800.0 PL=0
MOVL C00043 V=800.0 PL=0
MOVL C00044 V=800.0 PL=0
MOVL C00045 V=800.0 PL=0
MOVL C00046 V=800.0 PL=0
MOVL C00047 V=800.0 PL=0
MOVL C00048 V=800.0 PL=0
MOVL C00049 V=800.0 PL=0
MOVL C00050 V=800.0 PL=0
MOVL C00051 V=800.0 PL=0
MOVL C00052 V=800.0 PL=0
MOVL C00053 V=800.0 PL=0
MOVL C00054 V=800.0 PL=0
MOVL C00055 V=800.0 PL=0
MOVL C00056 V=800.0 PL=0
MOVL C00057 V=800.0 PL=0
MOVL C00058 V=800.0 PL=0
MOVL C00059 V=800.0 PL=0
MOVL C00060 V=800.0 PL=0
MOVL C00061 V=800.0 PL=0
MOVL C00062 V=800.0 PL=0
MOVL C00063 V=800.0 PL=0
MOVL C00064 V=800.0 PL=0
MOVL C00065 V=800.0 PL=0
MOVL C00066 V=800.0 PL=0
MOVL C00067 V=800.0 PL=0
MOVL C00068 V=800.0 PL=0
MOVL C00069 V=800.0 PL=0
MOVL C00070 V=800.0 PL=0
MOVL C00071 V=800.0 PL=0
MOVL C00072 V=800.0 PL=0
MOVL C00073 V=800.0 PL=0
MOVL C00074 V=800.0 PL=0
MOVL C00075 V=800.0 PL=0
MOVL C00076 V=800.0 PL=0
MOVL C00077 V=800.0 PL=0
MOVL C00078 V=800.0 PL=0
MOVL C00079 V=800.0 PL=0
MOVL C00080 V=800.0 PL=0
MOVL C00081 V=800.0 PL=0
MOVL C00082 V=800.0 PL=0
MOVL C00083 V=800.0 PL=0
MOVL C00084 V=800.0 PL=0
MOVL C00085 V=800.0 PL=0
MOVL C00086 V=800.0 PL=0
MOVL C00087 V=800.0 PL=0
MOVL C00088 V=800.0 PL=0
MOVL C00089 V=800.0 PL=0
MOVL C00090 V=800.0 PL=0
MOVL C00091 V=800.0 PL=0
MOVL C00092 V=800.0 PL=0
MOVL C00093 V=800.0 PL=0
MOVL C00094 V=800.0 PL=0
MOVL C00095 V=800.0 PL=0
MOVL C00096 V=800.0 PL=0
MOVL C00097 V=800.0 PL=0
MOVL C00098 V=800.0 PL=0
MOVL C00099 V=800.0 PL=0
MOVL C00100 V=800.0 PL=0
MOVL C00101 V=800.0 PL=0
MOVL C00102 V=800.0 PL=0
MOVL C00103 V=800.0 PL=0
MOVL C00104 V=800.0 PL=0
MOVL C00105 V=800.0 PL=0
MOVL C00106 V=800.0 PL=0
MOVL C00107 V=800.0 PL=0
MOVL C00108 V=800.0 PL=0
MOVL C00109 V=800.0 PL=0
MOVL C00110 V=800.0 PL=0
MOVL C00111 V=800.0 PL=0
MOVL C00112 V=800.0 PL=0
MOVL C00113 V=800.0 PL=0
MOVL C00114 V=800.0 PL=0
MOVL C00115 V=800.0 PL=0
MOVL C00116 V=800.0 PL=0
MOVL C00117 V=800.0 PL=0
MOVL C00118 V=800.0 PL=0
MOVL C00119 V=800.0 PL=0
MOVL C00120 V=800.0 PL=0
MOVL C00121 V=800.0 PL=0
MOVL C00122 V=800.0 PL=0
MOVL C00123 V=800.0 PL=0
MOVL C00124 V=800.0 PL=0
MOVL C00125 V=800.0 PL=0
MOVL C00126 V=800.0 PL=0
MOVL C00127 V=800.0 PL=0
MOVL C00128 V=800.0 PL=0
MOVL C00129 V=800.0 PL=0
MOVL C00130 V=800.0 PL=0
MOVL C00131 V=800.0 PL=0
MOVL C00132 V=800.0 PL=0
MOVL C00133 V=800.0 PL=0
MOVL C00134 V=800.0 PL=0
MOVL C00135 V=800.0 PL=0
MOVL C00136 V=800.0 PL=0
MOVL C00137 V=800.0 PL=0
MOVL C00138 V=800.0 PL=0
MOVL C00139 V=800.0 PL=0
MOVL C00140 V=800.0 PL=0
MOVL C00141 V=800.0 PL=0
MOVL C00142 V=800.0 PL=0
MOVL C00143 V=800.0 PL=0
MOVL C00144 V=800.0 PL=0
MOVL C00145 V=800.0 PL=0
MOVL C00146 V=800.0 PL=0
MOVL C00147 V=800.0 PL=0
MOVL C00148 V=800.0 PL=0
MOVL C00149 V=800.0 PL=0
MOVL C00150 V=800.0 PL=0
MOVL C00151 V=800.0 PL=0
MOVL C00152 V=800.0 PL=0
MOVL C00153 V=800.0 PL=0
MOVL C00154 V=800.0 PL=0
MOVL C00155 V=800.0 PL=0
MOVL C00156 V=800.0 PL=0
MOVL C00157 V=800.0 PL=0
MOVL C00158 V=800.0 PL=0
MOVL C00159 V=800.0 PL=0
MOVL C00160 V=800.0 PL=0
MOVL C00161 V=800.0 PL=0
MOVL C00162 V=800.0 PL=0
MOVL C00163 V=800.0 PL=0
MOVL C00164 V=800.0 PL=0
MOVL C00165 V=800.0 PL=0
MOVL C00166 V=800.0 PL=0
MOVL C00167 V=800.0 PL=0
MOVL C00168 V=800.0 PL=0
MOVL C00169 V=800.0 PL=0
MOVL C00170 V=800.0 PL=0
MOVL C00171 V=800.0 PL=0
MOVL C00172 V=800.0 PL=0
MOVL C00173 V=800.0 PL=0
MOVL C00174 V=800.0 PL=0
MOVL C00175 V=800.0 PL=0
MOVL C00176 V=800.0 PL=0
MOVL C00177 V=800.0 PL=0
MOVL C00178 V=800.0 PL=0
MOVL C00179 V=800.0 PL=0
MOVL C00180 V=800.0 PL=0
MOVL C00181 V=800.0 PL=0
MOVL C00182 V=800.0 PL=0
MOVL C00183 V=800.0 PL=0
MOVL C00184 V=800.0 PL=0
MOVL C00185 V=800.0 PL=0
MOVL C00186 V=800.0 PL=0
MOVL C00187 V=800.0 PL=0
MOVL C00188 V=800.0 PL=0
MOVL C00189 V=800.0 PL=0
MOVL C00190 V=800.0 PL=0
MOVL C00191 V=800.0 PL=0
MOVL C00192 V=800.0 PL=0
MOVL C00193 V=800.0 PL=0
MOVL C00194 V=800.0 PL=0
MOVL C00195 V=800.0 PL=0
MOVL C00196 V=800.0 PL=0
MOVL C00197 V=800.0 PL=0
MOVL C00198 V=800.0 PL=0
MOVL C00199 V=800.0 PL=0
MOVL C00200 V=800.0 PL=0
MOVL C00201 V=800.0 PL=0
MOVL C00202 V=800.0 PL=0
MOVL C00203 V=800.0 PL=0
MOVL C00204 V=800.0 PL=0
MOVL C00205 V=800.0 PL=0
MOVL C00206 V=800.0 PL=0
MOVL C00207 V=800.0 PL=0
MOVL C00208 V=800.0 PL=0
MOVL C00209 V=800.0 PL=0
MOVL C00210 V=800.0 PL=0
MOVL C00211 V=800.0 PL=0
MOVL C00212 V=800.0 PL=0
MOVL C00213 V=800.0 PL=0
MOVL C00214 V=800.0 PL=0
MOVL C00215 V=800.0 PL=0
MOVL C00216 V=800.0 PL=0
MOVL C00217 V=800.0 PL=0
MOVL C00218 V=800.0 PL=0
MOVL C00219 V=800.0 PL=0
MOVL C00220 V=800.0 PL=0
MOVL C00221 V=800.0 PL=0
MOVL C00222 V=800.0 PL=0
MOVL C00223 V=800.0 PL=0
MOVL C00224 V=800.0 PL=0
MOVL C00225 V=800.0 PL=0
MOVL C00226 V=800.0 PL=0
MOVL C00227 V=800.0 PL=0
MOVL C00228 V=800.0 PL=0
MOVL C00229 V=800.0 PL=0
MOVL C00230 V=800.0 PL=0
MOVL C00231 V=800.0 PL=0
MOVL C00232 V=800.0 PL=0
MOVL C00233 V=800.0 PL=0
MOVL C00234 V=800.0 PL=0
MOVL C00235 V=800.0 PL=0
MOVL C00236 V=800.0 PL=0
MOVL C00237 V=800.0 PL=0
MOVL C00238 V=800.0 PL=0
MOVL C00239 V=800.0 PL=0
MOVL C00240 V=800.0 PL=0
MOVL C00241 V=800.0 PL=0
MOVL C00242 V=800.0 PL=0
MOVL C00243 V=800.0 PL=0
MOVL C00244 V=800.0 PL=0
MOVL C00245 V=800.0 PL=0
MOVL C00246 V=800.0 PL=0
MOVL C00247 V=800.0 PL=0
MOVL C00248 V=800.0 PL=0
MOVL C00249 V=800.0 PL=0
MOVL C00250 V=800.0 PL=0
MOVL C00251 V=800.0 PL=0
MOVL C00252 V=800.0 PL=0
MOVL C00253 V=800.0 PL=0
MOVL C00254 V=800.0 PL=0
MOVL C00255 V=800.0 PL=0
MOVL C00256 V=800.0 PL=0
MOVL C00257 V=800.0 PL=0
MOVL C00258 V=800.0 PL=0
MOVL C00259 V=800.0 PL=0
MOVL C00260 V=800.0 PL=0
MOVL C00261 V=800.0 PL=0
MOVL C00262 V=800.0 PL=0
MOVL C00263 V=800.0 PL=0
MOVL C00264 V=800.0 PL=0
MOVL C00265 V=800.0 PL=0
MOVL C00266 V=800.0 PL=0
MOVL C00267 V=800.0 PL=0
MOVL C00268 V=800.0 PL=0
MOVL C00269 V=800.0 PL=0
MOVL C00270 V=800.0 PL=0
MOVL C00271 V=800.0 PL=0
MOVL C00272 V=800.0 PL=0
MOVL C00273 V=800.0 PL=0
MOVL C00274 V=800.0 PL=0
MOVL C00275 V=800.0 PL=0
MOVL C00276 V=800.0 PL=0
MOVL C00277 V=800.0 PL=0
MOVL C00278 V=800.0 PL=0
MOVL C00279 V=800.0 PL=0
MOVL C00280 V=800.0 PL=0
MOVL C00281 V=800.0 PL=0
MOVL C00282 V=800.0 PL=0
MOVL C00283 V=800.0 PL=0
MOVL C00284 V=800.0 PL=0
MOVL C00285 V=800.0 PL=0
MOVL C00286 V=800.0 PL=0
MOVL C00287 V=800.0 PL=0
MOVL C00288 V=800.0 PL=0
MOVL C00289 V=800.0 PL=0
MOVL C00290 V=800.0 PL=0
MOVL C00291 V=800.0 PL=0
MOVL C00292 V=800.0 PL=0
MOVL C00293 V=800.0 PL=0
MOVL C00294 V=800.0 PL=0
MOVL C00295 V=800.0 PL=0
MOVL C00296 V=800.0 PL=0
MOVL C00297 V=800.0 PL=0
MOVL C00298 V=800.0 PL=0
MOVL C00299 V=800.0 PL=0
MOVL C00300 V=800.0 PL=0
MOVL C00301 V=800.0 PL=0
MOVL C00302 V=800.0 PL=0
MOVL C00303 V=800.0 PL=0
MOVL C00304 V=800.0 PL=0
MOVL C00305 V=800.0 PL=0
MOVL C00306 V=800.0 PL=0
MOVL C00307 V=800.0 PL=0
MOVL C00308 V=800.0 PL=0
MOVL C00309 V=800.0 PL=0
MOVL C00310 V=800.0 PL=0
MOVL C00311 V=800.0 PL=0
MOVL C00312 V=800.0 PL=0
MOVL C00313 V=800.0 PL=0
MOVL C00314 V=800.0 PL=0
MOVL C00315 V=800.0 PL=0
MOVL C00316 V=800.0 PL=0
MOVL C00317 V=800.0 PL=0
MOVL C00318 V=800.0 PL=0
MOVL C00319 V=800.0 PL=0
MOVL C00320 V=800.0 PL=0
MOVL C00321 V=800.0 PL=0
MOVL C00322 V=800.0 PL=0
MOVL C00323 V=800.0 PL=0
MOVL C00324 V=800.0 PL=0
MOVL C00325 V=800.0 PL=0
MOVL C00326 V=800.0 PL=0
MOVL C00327 V=800.0 PL=0
MOVL C00328 V=800.0 PL=0
MOVL C00329 V=800.0 PL=0
MOVL C00330 V=800.0 PL=0
MOVL C00331 V=800.0 PL=0
MOVL C00332 V=800.0 PL=0
MOVL C00333 V=800.0 PL=0
MOVL C00334 V=800.0 PL=0
MOVL C00335 V=800.0 PL=0
MOVL C00336 V=800.0 PL=0
MOVL C00337 V=800.0 PL=0
MOVL C00338 V=800.0 PL=0
MOVL C00339 V=800.0 PL=0
MOVL C00340 V=800.0 PL=0
MOVL C00341 V=800.0 PL=0
MOVL C00342 V=800.0 PL=0
MOVL C00343 V=800.0 PL=0
MOVL C00344 V=800.0 PL=0
MOVL C00345 V=800.0 PL=0
MOVL C00346 V=800.0 PL=0
MOVL C00347 V=800.0 PL=0
MOVL C00348 V=800.0 PL=0
MOVL C00349 V=800.0 PL=0
MOVL C00350 V=800.0 PL=0
MOVL C00351 V=800.0 PL=0
MOVL C00352 V=800.0 PL=0
MOVL C00353 V=800.0 PL=0
MOVL C00354 V=800.0 PL=0
MOVL C00355 V=800.0 PL=0
MOVL C00356 V=800.0 PL=0
MOVL C00357 V=800.0 PL=0
MOVL C00358 V=800.0 PL=0
MOVL C00359 V=800.0 PL=0
MOVL C00360 V=800.0 PL=0
MOVL C00361 V=800.0 PL=0
MOVL C00362 V=800.0 PL=0
MOVL C00363 V=800.0 PL=0
MOVL C00364 V=800.0 PL=0
MOVL C00365 V=800.0 PL=0
MOVL C00366 V=800.0 PL=0
MOVL C00367 V=800.0 PL=0
MOVL C00368 V=800.0 PL=0
MOVL C00369 V=800.0 PL=0
MOVL C00370 V=800.0 PL=0
MOVL C00371 V=800.0 PL=0
MOVL C00372 V=800.0 PL=0
MOVL C00373 V=800.0 PL=0
MOVL C00374 V=800.0 PL=0
MOVL C00375 V=800.0 PL=0
MOVL C00376 V=800.0 PL=0
MOVL C00377 V=800.0 PL=0
MOVL C00378 V=800.0 PL=0
MOVL C00379 V=800.0 PL=0
MOVL C00380 V=800.0 PL=0
MOVL C00381 V=800.0 PL=0
MOVL C00382 V=800.0 PL=0
MOVL C00383 V=800.0 PL=0
MOVL C00384 V=800.0 PL=0
MOVL C00385 V=800.0 PL=0
MOVL C00386 V=800.0 PL=0
MOVL C00387 V=800.0 PL=0
MOVL C00388 V=800.0 PL=0
MOVL C00389 V=800.0 PL=0
MOVL C00390 V=800.0 PL=0
MOVL C00391 V=800.0 PL=0
MOVL C00392 V=800.0 PL=0
MOVL C00393 V=800.0 PL=0
MOVL C00394 V=800.0 PL=0
MOVL C00395 V=800.0 PL=0
MOVL C00396 V=800.0 PL=0
MOVL C00397 V=800.0 PL=0
MOVL C00398 V=800.0 PL=0
MOVL C00399 V=800.0 PL=0
MOVL C00400 V=800.0 PL=0
MOVL C00401 V=800.0 PL=0
MOVL C00402 V=800.0 PL=0
MOVL C00403 V=800.0 PL=0
MOVL C00404 V=800.0 PL=0
MOVL C00405 V=800.0 PL=0
MOVL C00406 V=800.0 PL=0
MOVL C00407 V=800.0 PL=0
MOVL C00408 V=800.0 PL=0
MOVL C00409 V=800.0 PL=0
MOVL C00410 V=800.0 PL=0
MOVL C00411 V=800.0 PL=0
MOVL C00412 V=800.0 PL=0
MOVL C00413 V=800.0 PL=0
MOVL C00414 V=800.0 PL=0
MOVL C00415 V=800.0 PL=0
MOVL C00416 V=800.0 PL=0
MOVL C00417 V=800.0 PL=0
MOVL C00418 V=800.0 PL=0
MOVL C00419 V=800.0 PL=0
MOVL C00420 V=800.0 PL=0
MOVL C00421 V=800.0 PL=0
MOVL C00422 V=800.0 PL=0
MOVL C00423 V=800.0 PL=0
MOVL C00424 V=800.0 PL=0
MOVL C00425 V=800.0 PL=0
MOVL C00426 V=800.0 PL=0
MOVL C00427 V=800.0 PL=0
MOVL C00428 V=800.0 PL=0
MOVL C00429 V=800.0 PL=0
MOVL C00430 V=800.0 PL=0
MOVL C00431 V=800.0 PL=0
MOVL C00432 V=800.0 PL=0
MOVL C00433 V=800.0 PL=0
MOVL C00434 V=800.0 PL=0
MOVL C00435 V=800.0 PL=0
MOVL C00436 V=800.0 PL=0
MOVL C00437 V=800.0 PL=0
MOVL C00438 V=800.0 PL=0
MOVL C00439 V=800.0 PL=0
MOVL C00440 V=800.0 PL=0
MOVL C00441 V=800.0 PL=0
MOVL C00442 V=800.0 PL=0
MOVL C00443 V=800.0 PL=0
MOVL C00444 V=800.0 PL=0
MOVL C00445 V=800.0 PL=0
MOVL C00446 V=800.0 PL=0
MOVL C00447 V=800.0 PL=0
MOVL C00448 V=800.0 PL=0
MOVL C00449 V=800.0 PL=0
MOVL C00450 V=800.0 PL=0
MOVL C00451 V=800.0 PL=0
MOVL C00452 V=800.0 PL=0
MOVL C00453 V=800.0 PL=0
MOVL C00454 V=800.0 PL=0
MOVL C00455 V=800.0 PL=0
MOVL C00456 V=800.0 PL=0
MOVL C00457 V=800.0 PL=0
MOVL C00458 V=800.0 PL=0
MOVL C00459 V=800.0 PL=0
MOVL C00460 V=800.0 PL=0
MOVL C00461 V=800.0 PL=0
MOVL C00462 V=800.0 PL=0
MOVL C00463 V=800.0 PL=0
MOVL C00464 V=800.0 PL=0
MOVL C00465 V=800.0 PL=0
MOVL C00466 V=800.0 PL=0
MOVL C00467 V=800.0 PL=0
MOVL C00468 V=800.0 PL=0
MOVL C00469 V=800.0 PL=0
MOVL C00470 V=800.0 PL=0
MOVL C00471 V=800.0 PL=0
MOVL C00472 V=800.0 PL=0
MOVL C00473 V=800.0 PL=0
MOVL C00474 V=800.0 PL=0
MOVL C00475 V=800.0 PL=0
MOVL C00476 V=800.0 PL=0
MOVL C00477 V=800.0 PL=0
MOVL C00478 V=800.0 PL=0
MOVL C00479 V=800.0 PL=0
MOVL C00480 V=800.0 PL=0
MOVL C00481 V=800.0 PL=0
MOVL C00482 V=800.0 PL=0
MOVL C00483 V=800.0 PL=0
MOVL C00484 V=800.0 PL=0
MOVL C00485 V=800.0 PL=0
MOVL C00486 V=800.0 PL=0
MOVL C00487 V=800.0 PL=0
MOVL C00488 V=800.0 PL=0
MOVL C00489 V=800.0 PL=0
MOVL C00490 V=800.0 PL=0
MOVL C00491 V=800.0 PL=0
MOVL C00492 V=800.0 PL=0
MOVL C00493 V=800.0 PL=0
MOVL C00494 V=800.0 PL=0
MOVL C00495 V=800.0 PL=0
MOVL C00496 V=800.0 PL=0
MOVL C00497 V=800.0 PL=0
MOVL C00498 V=800.0 PL=0
MOVL C00499 V=800.0 PL=0
MOVL C00500 V=800.0 PL=0
MOVL C00501 V=800.0 PL=0
MOVL C00502 V=800.0 PL=0
MOVL C00503 V=800.0 PL=0
MOVL C00504 V=800.0 PL=0
MOVL C00505 V=800.0 PL=0
MOVL C00506 V=800.0 PL=0
MOVL C00507 V=800.0 PL=0
MOVL C00508 V=800.0 PL=0
MOVL C00509 V=800.0 PL=0
MOVL C00510 V=800.0 PL=0
MOVL C00511 V=800.0 PL=0
MOVL C00512 V=800.0 PL=0
MOVL C00513 V=800.0 PL=0
MOVL C00514 V=800.0 PL=0
MOVL C00515 V=800.0 PL=0
MOVL C00516 V=800.0 PL=0
MOVL C00517 V=800.0 PL=0
MOVL C00518 V=800.0 PL=0
MOVL C00519 V=800.0 PL=0
MOVL C00520 V=800.0 PL=0
MOVL C00521 V=800.0 PL=0
MOVL C00522 V=800.0 PL=0
MOVL C00523 V=800.0 PL=0
MOVL C00524 V=800.0 PL=0
MOVL C00525 V=800.0 PL=0
MOVL C00526 V=800.0 PL=0
MOVL C00527 V=800.0 PL=0
MOVL C00528 V=800.0 PL=0
MOVL C00529 V=800.0 PL=0
MOVL C00530 V=800.0 PL=0
MOVL C00531 V=800.0 PL=0
MOVL C00532 V=800.0 PL=0
MOVL C00533 V=800.0 PL=0
MOVL C00534 V=800.0 PL=0
MOVL C00535 V=800.0 PL=0
MOVL C00536 V=800.0 PL=0
MOVL C00537 V=800.0 PL=0
MOVL C00538 V=800.0 PL=0
MOVL C00539 V=800.0 PL=0
MOVL C00540 V=800.0 PL=0
MOVL C00541 V=800.0 PL=0
MOVL C00542 V=800.0 PL=0
MOVL C00543 V=800.0 PL=0
MOVL C00544 V=800.0 PL=0
MOVL C00545 V=800.0 PL=0
MOVL C00546 V=800.0 PL=0
MOVL C00547 V=800.0 PL=0
MOVL C00548 V=800.0 PL=0
MOVL C00549 V=800.0 PL=0
MOVL C00550 V=800.0 PL=0
MOVL C00551 V=800.0 PL=0
MOVL C00552 V=800.0 PL=0
MOVL C00553 V=800.0 PL=0
MOVL C00554 V=800.0 PL=0
MOVL C00555 V=800.0 PL=0
MOVL C00556 V=800.0 PL=0
MOVL C00557 V=800.0 PL=0
MOVL C00558 V=800.0 PL=0
MOVL C00559 V=800.0 PL=0
MOVL C00560 V=800.0 PL=0
MOVL C00561 V=800.0 PL=0
MOVL C00562 V=800.0 PL=0
MOVL C00563 V=800.0 PL=0
MOVL C00564 V=800.0 PL=0
MOVL C00565 V=800.0 PL=0
MOVL C00566 V=800.0 PL=0
MOVL C00567 V=800.0 PL=0
MOVL C00568 V=800.0 PL=0
MOVL C00569 V=800.0 PL=0
MOVL C00570 V=800.0 PL=0
MOVL C00571 V=800.0 PL=0
MOVL C00572 V=800.0 PL=0
MOVL C00573 V=800.0 PL=0
MOVL C00574 V=800.0 PL=0
MOVL C00575 V=800.0 PL=0
MOVL C00576 V=800.0 PL=0
MOVL C00577 V=800.0 PL=0
MOVL C00578 V=800.0 PL=0
MOVL C00579 V=800.0 PL=0
MOVL C00580 V=800.0 PL=0
MOVL C00581 V=800.0 PL=0
MOVL C00582 V=800.0 PL=0
MOVL C00583 V=800.0 PL=0
MOVL C00584 V=800.0 PL=0
MOVL C00585 V=800.0 PL=0
MOVL C00586 V=800.0 PL=0
MOVL C00587 V=800.0 PL=0
MOVL C00588 V=800.0 PL=0
MOVL C00589 V=800.0 PL=0
MOVL C00590 V=800.0 PL=0
MOVL C00591 V=800.0 PL=0
MOVL C00592 V=800.0 PL=0
MOVL C00593 V=800.0 PL=0
MOVL C00594 V=800.0 PL=0
MOVL C00595 V=800.0 PL=0
MOVL C00596 V=800.0 PL=0
MOVL C00597 V=800.0 PL=0
MOVL C00598 V=800.0 PL=0
MOVL C00599 V=800.0 PL=0
MOVL C00600 V=800.0 PL=0
MOVL C00601 V=800.0 PL=0
MOVL C00602 V=800.0 PL=0
MOVL C00603 V=800.0 PL=0
MOVL C00604 V=800.0 PL=0
MOVL C00605 V=800.0 PL=0
MOVL C00606 V=800.0 PL=0
MOVL C00607 V=800.0 PL=0
MOVL C00608 V=800.0 PL=0
MOVL C00609 V=800.0 PL=0
MOVL C00610 V=800.0 PL=0
MOVL C00611 V=800.0 PL=0
MOVL C00612 V=800.0 PL=0
MOVL C00613 V=800.0 PL=0
MOVL C00614 V=800.0 PL=0
MOVL C00615 V=800.0 PL=0
MOVL C00616 V=800.0 PL=0
MOVL C00617 V=800.0 PL=0
MOVL C00618 V=800.0 PL=0
MOVL C00619 V=800.0 PL=0
MOVL C00620 V=800.0 PL=0
MOVL C00621 V=800.0 PL=0
MOVL C00622 V=800.0 PL=0
MOVL C00623 V=800.0 PL=0
MOVL C00624 V=800.0 PL=0
MOVL C00625 V=800.0 PL=0
MOVL C00626 V=800.0 PL=0
MOVL C00627 V=800.0 PL=0
MOVL C00628 V=800.0 PL=0
MOVL C00629 V=800.0 PL=0
MOVL C00630 V=800.0 PL=0
MOVL C00631 V=800.0 PL=0
MOVL C00632 V=800.0 PL=0
MOVL C00633 V=800.0 PL=0
MOVL C00634 V=800.0 PL=0
MOVL C00635 V=800.0 PL=0
MOVL C00636 V=800.0 PL=0
MOVL C00637 V=800.0 PL=0
MOVL C00638 V=800.0 PL=0
MOVL C00639 V=800.0 PL=0
MOVL C00640 V=800.0 PL=0
MOVL C00641 V=800.0 PL=0
MOVL C00642 V=800.0 PL=0
MOVL C00643 V=800.0 PL=0
MOVL C00644 V=800.0 PL=0
MOVL C00645 V=800.0 PL=0
MOVL C00646 V=800.0 PL=0
MOVL C00647 V=800.0 PL=0
MOVL C00648 V=800.0 PL=0
MOVL C00649 V=800.0 PL=0
MOVL C00650 V=800.0 PL=0
MOVL C00651 V=800.0 PL=0
MOVL C00652 V=800.0 PL=0
MOVL C00653 V=800.0 PL=0
MOVL C00654 V=800.0 PL=0
MOVL C00655 V=800.0 PL=0
MOVL C00656 V=800.0 PL=0
MOVL C00657 V=800.0 PL=0
MOVL C00658 V=800.0 PL=0
MOVL C00659 V=800.0 PL=0
MOVL C00660 V=800.0 PL=0
MOVL C00661 V=800.0 PL=0
MOVL C00662 V=800.0 PL=0
MOVL C00663 V=800.0 PL=0
MOVL C00664 V=800.0 PL=0
MOVL C00665 V=800.0 PL=0
MOVL C00666 V=800.0 PL=0
MOVL C00667 V=800.0 PL=0
MOVL C00668 V=800.0 PL=0
MOVL C00669 V=800.0 PL=0
MOVL C00670 V=800.0 PL=0
MOVL C00671 V=800.0 PL=0
MOVL C00672 V=800.0 PL=0
MOVL C00673 V=800.0 PL=0
MOVL C00674 V=800.0 PL=0
MOVL C00675 V=800.0 PL=0
MOVL C00676 V=800.0 PL=0
MOVL C00677 V=800.0 PL=0
MOVL C00678 V=800.0 PL=0
MOVL C00679 V=800.0 PL=0
MOVL C00680 V=800.0 PL=0
MOVL C00681 V=800.0 PL=0
MOVL C00682 V=800.0 PL=0
MOVL C00683 V=800.0 PL=0
MOVL C00684 V=800.0 PL=0
MOVL C00685 V=800.0 PL=0
MOVL C00686 V=800.0 PL=0
MOVL C00687 V=800.0 PL=0
MOVL C00688 V=800.0 PL=0
MOVL C00689 V=800.0 PL=0
MOVL C00690 V=800.0 PL=0
MOVL C00691 V=800.0 PL=0
MOVL C00692 V=800.0 PL=0
MOVL C00693 V=800.0 PL=0
MOVL C00694 V=800.0 PL=0
MOVL C00695 V=800.0 PL=0
MOVL C00696 V=800.0 PL=0
MOVL C00697 V=800.0 PL=0
MOVL C00698 V=800.0 PL=0
MOVL C00699 V=800.0 PL=0
MOVL C00700 V=800.0 PL=0
MOVL C00701 V=800.0 PL=0
MOVL C00702 V=800.0 PL=0
MOVL C00703 V=800.0 PL=0
MOVL C00704 V=800.0 PL=0
MOVL C00705 V=800.0 PL=0
MOVL C00706 V=800.0 PL=0
MOVL C00707 V=800.0 PL=0
MOVL C00708 V=800.0 PL=0
MOVL C00709 V=800.0 PL=0
MOVL C00710 V=800.0 PL=0
MOVL C00711 V=800.0 PL=0
MOVL C00712 V=800.0 PL=0
MOVL C00713 V=800.0 PL=0
MOVL C00714 V=800.0 PL=0
MOVL C00715 V=800.0 PL=0
MOVL C00716 V=800.0 PL=0
MOVL C00717 V=800.0 PL=0
MOVL C00718 V=800.0 PL=0
MOVL C00719 V=800.0 PL=0
MOVL C00720 V=800.0 PL=0
MOVL C00721 V=800.0 PL=0
MOVL C00722 V=800.0 PL=0
MOVL C00723 V=800.0 PL=0
MOVL C00724 V=800.0 PL=0
MOVL C00725 V=800.0 PL=0
MOVL C00726 V=800.0 PL=0
MOVL C00727 V=800.0 PL=0
MOVL C00728 V=800.0 PL=0
MOVL C00729 V=800.0 PL=0
MOVL C00730 V=800.0 PL=0
MOVL C00731 V=800.0 PL=0
MOVL C00732 V=800.0 PL=0
MOVL C00733 V=800.0 PL=0
MOVL C00734 V=800.0 PL=0
MOVL C00735 V=800.0 PL=0
MOVL C00736 V=800.0 PL=0
MOVL C00737 V=800.0 PL=0
MOVL C00738 V=800.0 PL=0
MOVL C00739 V=800.0 PL=0
MOVL C00740 V=800.0 PL=0
MOVL C00741 V=800.0 PL=0
MOVL C00742 V=800.0 PL=0
MOVL C00743 V=800.0 PL=0
MOVL C00744 V=800.0 PL=0
MOVL C00745 V=800.0 PL=0
MOVL C00746 V=800.0 PL=0
MOVL C00747 V=800.0 PL=0
MOVL C00748 V=800.0 PL=0
MOVL C00749 V=800.0 PL=0
MOVL C00750 V=800.0 PL=0
MOVL C00751 V=800.0 PL=0
MOVL C00752 V=800.0 PL=0
MOVL C00753 V=800.0 PL=0
MOVL C00754 V=800.0 PL=0
MOVL C00755 V=800.0 PL=0
MOVL C00756 V=800.0 PL=0
MOVL C00757 V=800.0 PL=0
MOVL C00758 V=800.0 PL=0
MOVL C00759 V=800.0 PL=0
MOVL C00760 V=800.0 PL=0
MOVL C00761 V=800.0 PL=0
MOVL C00762 V=800.0 PL=0
MOVL C00763 V=800.0 PL=0
MOVL C00764 V=800.0 PL=0
MOVL C00765 V=800.0 PL=0
MOVL C00766 V=800.0 PL=0
MOVL C00767 V=800.0 PL=0
MOVL C00768 V=800.0 PL=0
MOVL C00769 V=800.0 PL=0
MOVL C00770 V=800.0 PL=0
MOVL C00771 V=800.0 PL=0
MOVL C00772 V=800.0 PL=0
MOVL C00773 V=800.0 PL=0
MOVL C00774 V=800.0 PL=0
MOVL C00775 V=800.0 PL=0
MOVL C00776 V=800.0 PL=0
MOVL C00777 V=800.0 PL=0
MOVL C00778 V=800.0 PL=0
MOVL C00779 V=800.0 PL=0
MOVL C00780 V=800.0 PL=0
MOVL C00781 V=800.0 PL=0
MOVL C00782 V=800.0 PL=0
MOVL C00783 V=800.0 PL=0
MOVL C00784 V=800.0 PL=0
MOVL C00785 V=800.0 PL=0
MOVL C00786 V=800.0 PL=0
MOVL C00787 V=800.0 PL=0
MOVL C00788 V=800.0 PL=0
MOVL C00789 V=800.0 PL=0
MOVL C00790 V=800.0 PL=0
MOVL C00791 V=800.0 PL=0
MOVL C00792 V=800.0 PL=0
MOVL C00793 V=800.0 PL=0
MOVL C00794 V=800.0 PL=0
MOVL C00795 V=800.0 PL=0
MOVL C00796 V=800.0 PL=0
MOVL C00797 V=800.0 PL=0
MOVL C00798 V=800.0 PL=0
MOVL C00799 V=800.0 PL=0
MOVL C00800 V=800.0 PL=0
MOVL C00801 V=800.0 PL=0
MOVL C00802 V=800.0 PL=0
MOVL C00803 V=800.0 PL=0
MOVL C00804 V=800.0 PL=0
MOVL C00805 V=800.0 PL=0
MOVL C00806 V=800.0 PL=0
MOVL C00807 V=800.0 PL=0
MOVL C00808 V=800.0 PL=0
MOVL C00809 V=800.0 PL=0
MOVL C00810 V=800.0 PL=0
MOVL C00811 V=800.0 PL=0
MOVL C00812 V=800.0 PL=0
MOVL C00813 V=800.0 PL=0
MOVL C00814 V=800.0 PL=0
MOVL C00815 V=800.0 PL=0
MOVL C00816 V=800.0 PL=0
MOVL C00817 V=800.0 PL=0
MOVL C00818 V=800.0 PL=0
MOVL C00819 V=800.0 PL=0
MOVL C00820 V=800.0 PL=0
MOVL C00821 V=800.0 PL=0
MOVL C00822 V=800.0 PL=0
MOVL C00823 V=800.0 PL=0
MOVL C00824 V=800.0 PL=0
MOVL C00825 V=800.0 PL=0
MOVL C00826 V=800.0 PL=0
MOVL C00827 V=800.0 PL=0
MOVL C00828 V=800.0 PL=0
MOVL C00829 V=800.0 PL=0
MOVL C00830 V=800.0 PL=0
MOVL C00831 V=800.0 PL=0
MOVL C00832 V=800.0 PL=0
MOVL C00833 V=800.0 PL=0
MOVL C00834 V=800.0 PL=0
MOVL C00835 V=800.0 PL=0
MOVL C00836 V=800.0 PL=0
MOVL C00837 V=800.0 PL=0
MOVL C00838 V=800.0 PL=0
MOVL C00839 V=800.0 PL=0
MOVL C00840 V=800.0 PL=0
MOVL C00841 V=800.0 PL=0
MOVL C00842 V=800.0 PL=0
MOVL C00843 V=800.0 PL=0
MOVL C00844 V=800.0 PL=0
MOVL C00845 V=800.0 PL=0
MOVL C00846 V=800.0 PL=0
MOVL C00847 V=800.0 PL=0
MOVL C00848 V=800.0 PL=0
MOVL C00849 V=800.0 PL=0
MOVL C00850 V=800.0 PL=0
MOVL C00851 V=800.0 PL=0
MOVL C00852 V=800.0 PL=0
MOVL C00853 V=800.0 PL=0
MOVL C00854 V=800.0 PL=0
MOVL C00855 V=800.0 PL=0
MOVL C00856 V=800.0 PL=0
MOVL C00857 V=800.0 PL=0
MOVL C00858 V=800.0 PL=0
MOVL C00859 V=800.0 PL=0
MOVL C00860 V=800.0 PL=0
MOVL C00861 V=800.0 PL=0
MOVL C00862 V=800.0 PL=0
MOVL C00863 V=800.0 PL=0
MOVL C00864 V=800.0 PL=0
MOVL C00865 V=800.0 PL=0
MOVL C00866 V=800.0 PL=0
MOVL C00867 V=800.0 PL=0
MOVL C00868 V=800.0 PL=0
MOVL C00869 V=800.0 PL=0
MOVL C00870 V=800.0 PL=0
MOVL C00871 V=800.0 PL=0
MOVL C00872 V=800.0 PL=0
MOVL C00873 V=800.0 PL=0
MOVL C00874 V=800.0 PL=0
MOVL C00875 V=800.0 PL=0
MOVL C00876 V=800.0 PL=0
MOVL C00877 V=800.0 PL=0
MOVL C00878 V=800.0 PL=0
MOVL C00879 V=800.0 PL=0
MOVL C00880 V=800.0 PL=0
MOVL C00881 V=800.0 PL=0
MOVL C00882 V=800.0 PL=0
MOVL C00883 V=800.0 PL=0
MOVL C00884 V=800.0 PL=0
MOVL C00885 V=800.0 PL=0
MOVL C00886 V=800.0 PL=0
MOVL C00887 V=800.0 PL=0
MOVL C00888 V=800.0 PL=0
MOVL C00889 V=800.0 PL=0
MOVL C00890 V=800.0 PL=0
MOVL C00891 V=800.0 PL=0
MOVL C00892 V=800.0 PL=0
MOVL C00893 V=800.0 PL=0
MOVL C00894 V=800.0 PL=0
MOVL C00895 V=800.0 PL=0
MOVL C00896 V=800.0 PL=0
MOVL C00897 V=800.0 PL=0
MOVL C00898 V=800.0 PL=0
MOVL C00899 V=800.0 PL=0
MOVL C00900 V=800.0 PL=0
MOVL C00901 V=800.0 PL=0
MOVL C00902 V=800.0 PL=0
MOVL C00903 V=800.0 PL=0
MOVL C00904 V=800.0 PL=0
MOVL C00905 V=800.0 PL=0
MOVL C00906 V=800.0 PL=0
MOVL C00907 V=800.0 PL=0
MOVL C00908 V=800.0 PL=0
MOVL C00909 V=800.0 PL=0
MOVL C00910 V=800.0 PL=0
MOVL C00911 V=800.0 PL=0
MOVL C00912 V=800.0 PL=0
MOVL C00913 V=800.0 PL=0
MOVL C00914 V=800.0 PL=0
MOVL C00915 V=800.0 PL=0
MOVL C00916 V=800.0 PL=0
MOVL C00917 V=800.0 PL=0
MOVL C00918 V=800.0 PL=0
MOVL C00919 V=800.0 PL=0
MOVL C00920 V=800.0 PL=0
MOVL C00921 V=800.0 PL=0
MOVL C00922 V=800.0 PL=0
MOVL C00923 V=800.0 PL=0
MOVL C00924 V=800.0 PL=0
MOVL C00925 V=800.0 PL=0
MOVL C00926 V=800.0 PL=0
MOVL C00927 V=800.0 PL=0
MOVL C00928 V=800.0 PL=0
MOVL C00929 V=800.0 PL=0
MOVL C00930 V=800.0 PL=0
MOVL C00931 V=800.0 PL=0
MOVL C00932 V=800.0 PL=0
MOVL C00933 V=800.0 PL=0
MOVL C00934 V=800.0 PL=0
MOVL C00935 V=800.0 PL=0
MOVL C00936 V=800.0 PL=0
MOVL C00937 V=800.0 PL=0
MOVL C00938 V=800.0 PL=0
MOVL C00939 V=800.0 PL=0
MOVL C00940 V=800.0 PL=0
MOVL C00941 V=800.0 PL=0
MOVL C00942 V=800.0 PL=0
MOVL C00943 V=800.0 PL=0
MOVL C00944 V=800.0 PL=0
MOVL C00945 V=800.0 PL=0
MOVL C00946 V=800.0 PL=0
MOVL C00947 V=800.0 PL=0
MOVL C00948 V=800.0 PL=0
MOVL C00949 V=800.0 PL=0
MOVL C00950 V=800.0 PL=0
MOVL C00951 V=800.0 PL=0
MOVL C00952 V=800.0 PL=0
MOVL C00953 V=800.0 PL=0
MOVL C00954 V=800.0 PL=0
MOVL C00955 V=800.0 PL=0
MOVL C00956 V=800.0 PL=0
MOVL C00957 V=800.0 PL=0
MOVL C00958 V=800.0 PL=0
MOVL C00959 V=800.0 PL=0
MOVL C00960 V=800.0 PL=0
MOVL C00961 V=800.0 PL=0
MOVL C00962 V=800.0 PL=0
MOVL C00963 V=800.0 PL=0
MOVL C00964 V=800.0 PL=0
MOVL C00965 V=800.0 PL=0
MOVL C00966 V=800.0 PL=0
MOVL C00967 V=800.0 PL=0
MOVL C00968 V=800.0 PL=0
MOVL C00969 V=800.0 PL=0
MOVL C00970 V=800.0 PL=0
MOVL C00971 V=800.0 PL=0
MOVL C00972 V=800.0 PL=0
MOVL C00973 V=800.0 PL=0
MOVL C00974 V=800.0 PL=0
MOVL C00975 V=800.0 PL=0
MOVL C00976 V=800.0 PL=0
MOVL C00977 V=800.0 PL=0
MOVL C00978 V=800.0 PL=0
MOVL C00979 V=800.0 PL=0
MOVL C00980 V=800.0 PL=0
MOVL C00981 V=800.0 PL=0
MOVL C00982 V=800.0 PL=0
MOVL C00983 V=800.0 PL=0
MOVL C00984 V=800.0 PL=0
MOVL C00985 V=800.0 PL=0
MOVL C00986 V=800.0 PL=0
MOVL C00987 V=800.0 PL=0
MOVL C00988 V=800.0 PL=0
MOVL C00989 V=800.0 PL=0
MOVL C00990 V=800.0 PL=0
MOVL C00991 V=800.0 PL=0
MOVL C00992 V=800.0 PL=0
MOVL C00993 V=800.0 PL=0
MOVL C00994 V=800.0 PL=0
MOVL C00995 V=800.0 PL=0
MOVL C00996 V=800.0 PL=0
MOVL C00997 V=800.0 PL=0
MOVL C00998 V=800.0 PL=0
MOVL C00999 V=800.0 PL=0
MOVL C01000 V=800.0 PL=0
MOVL C01001 V=800.0 PL=0
MOVL C01002 V=800.0 PL=0
MOVL C01003 V=800.0 PL=0
MOVL C01004 V=800.0 PL=0
MOVL C01005 V=800.0 PL=0
MOVL C01006 V=800.0 PL=0
MOVL C01007 V=800.0 PL=0
MOVL C01008 V=800.0 PL=0
MOVL C01009 V=800.0 PL=0
MOVL C01010 V=800.0 PL=0
MOVL C01011 V=800.0 PL=0
MOVL C01012 V=800.0 PL=0
MOVL C01013 V=800.0 PL=0
MOVL C01014 V=800.0 PL=0
MOVL C01015 V=800.0 PL=0
MOVL C01016 V=800.0 PL=0
MOVL C01017 V=800.0 PL=0
MOVL C01018 V=800.0 PL=0
MOVL C01019 V=800.0 PL=0
MOVL C01020 V=800.0 PL=0
MOVL C01021 V=800.0 PL=0
MOVL C01022 V=800.0 PL=0
MOVL C01023 V=800.0 PL=0
MOVL C01024 V=800.0 PL=0
MOVL C01025 V=800.0 PL=0
MOVL C01026 V=800.0 PL=0
MOVL C01027 V=800.0 PL=0
MOVL C01028 V=800.0 PL=0
MOVL C01029 V=800.0 PL=0
MOVL C01030 V=800.0 PL=0
MOVL C01031 V=800.0 PL=0
MOVL C01032 V=800.0 PL=0
MOVL C01033 V=800.0 PL=0
MOVL C01034 V=800.0 PL=0
MOVL C01035 V=800.0 PL=0
MOVL C01036 V=800.0 PL=0
MOVL C01037 V=800.0 PL=0
MOVL C01038 V=800.0 PL=0
MOVL C01039 V=800.0 PL=0
MOVL C01040 V=800.0 PL=0
MOVL C01041 V=800.0 PL=0
MOVL C01042 V=800.0 PL=0
MOVL C01043 V=800.0 PL=0
MOVL C01044 V=800.0 PL=0
MOVL C01045 V=800.0 PL=0
MOVL C01046 V=800.0 PL=0
MOVL C01047 V=800.0 PL=0
MOVL C01048 V=800.0 PL=0
MOVL C01049 V=800.0 PL=0
MOVL C01050 V=800.0 PL=0
MOVL C01051 V=800.0 PL=0
MOVL C01052 V=800.0 PL=0
MOVL C01053 V=800.0 PL=0
MOVL C01054 V=800.0 PL=0
MOVL C01055 V=800.0 PL=0
MOVL C01056 V=800.0 PL=0
MOVL C01057 V=800.0 PL=0
MOVL C01058 V=800.0 PL=0
MOVL C01059 V=800.0 PL=0
MOVL C01060 V=800.0 PL=0
MOVL C01061 V=800.0 PL=0
MOVL C01062 V=800.0 PL=0
MOVL C01063 V=800.0 PL=0
MOVL C01064 V=800.0 PL=0
MOVL C01065 V=800.0 PL=0
MOVL C01066 V=800.0 PL=0
MOVL C01067 V=800.0 PL=0
MOVL C01068 V=800.0 PL=0
MOVL C01069 V=800.0 PL=0
MOVL C01070 V=800.0 PL=0
MOVL C01071 V=800.0 PL=0
MOVL C01072 V=800.0 PL=0
MOVL C01073 V=800.0 PL=0
MOVL C01074 V=800.0 PL=0
MOVL C01075 V=800.0 PL=0
MOVL C01076 V=800.0 PL=0
MOVL C01077 V=800.0 PL=0
MOVL C01078 V=800.0 PL=0
MOVL C01079 V=800.0 PL=0
MOVL C01080 V=800.0 PL=0
MOVL C01081 V=800.0 PL=0
MOVL C01082 V=800.0 PL=0
MOVL C01083 V=800.0 PL=0
MOVL C01084 V=800.0 PL=0
MOVL C01085 V=800.0 PL=0
MOVL C01086 V=800.0 PL=0
MOVL C01087 V=800.0 PL=0
MOVL C01088 V=800.0 PL=0
MOVL C01089 V=800.0 PL=0
MOVL C01090 V=800.0 PL=0
MOVL C01091 V=800.0 PL=0
MOVL C01092 V=800.0 PL=0
MOVL C01093 V=800.0 PL=0
MOVL C01094 V=800.0 PL=0
MOVL C01095 V=800.0 PL=0
MOVL C01096 V=800.0 PL=0
MOVL C01097 V=800.0 PL=0
MOVL C01098 V=800.0 PL=0
MOVL C01099 V=800.0 PL=0
MOVL C01100 V=800.0 PL=0
MOVL C01101 V=800.0 PL=0
MOVL C01102 V=800.0 PL=0
MOVL C01103 V=800.0 PL=0
MOVL C01104 V=800.0 PL=0
MOVL C01105 V=800.0 PL=0
MOVL C01106 V=800.0 PL=0
MOVL C01107 V=800.0 PL=0
MOVL C01108 V=800.0 PL=0
MOVL C01109 V=800.0 PL=0
MOVL C01110 V=800.0 PL=0
MOVL C01111 V=800.0 PL=0
MOVL C01112 V=800.0 PL=0
MOVL C01113 V=800.0 PL=0
MOVL C01114 V=800.0 PL=0
MOVL C01115 V=800.0 PL=0
MOVL C01116 V=800.0 PL=0
MOVL C01117 V=800.0 PL=0
MOVL C01118 V=800.0 PL=0
MOVL C01119 V=800.0 PL=0
MOVL C01120 V=800.0 PL=0
MOVL C01121 V=800.0 PL=0
MOVL C01122 V=800.0 PL=0
MOVL C01123 V=800.0 PL=0
MOVL C01124 V=800.0 PL=0
MOVL C01125 V=800.0 PL=0
MOVL C01126 V=800.0 PL=0
MOVL C01127 V=800.0 PL=0
MOVL C01128 V=800.0 PL=0
MOVL C01129 V=800.0 PL=0
MOVL C01130 V=800.0 PL=0
MOVL C01131 V=800.0 PL=0
MOVL C01132 V=800.0 PL=0
MOVL C01133 V=800.0 PL=0
MOVL C01134 V=800.0 PL=0
MOVL C01135 V=800.0 PL=0
MOVL C01136 V=800.0 PL=0
MOVL C01137 V=800.0 PL=0
MOVL C01138 V=800.0 PL=0
MOVL C01139 V=800.0 PL=0
MOVL C01140 V=800.0 PL=0
MOVL C01141 V=800.0 PL=0
MOVL C01142 V=800.0 PL=0
MOVL C01143 V=800.0 PL=0
MOVL C01144 V=800.0 PL=0
MOVL C01145 V=800.0 PL=0
MOVL C01146 V=800.0 PL=0
MOVL C01147 V=800.0 PL=0
MOVL C01148 V=800.0 PL=0
MOVL C01149 V=800.0 PL=0
MOVL C01150 V=800.0 PL=0
MOVL C01151 V=800.0 PL=0
MOVL C01152 V=800.0 PL=0
MOVL C01153 V=800.0 PL=0
MOVL C01154 V=800.0 PL=0
MOVL C01155 V=800.0 PL=0
MOVL C01156 V=800.0 PL=0
MOVL C01157 V=800.0 PL=0
MOVL C01158 V=800.0 PL=0
MOVL C01159 V=800.0 PL=0
MOVL C01160 V=800.0 PL=0
MOVL C01161 V=800.0 PL=0
MOVL C01162 V=800.0 PL=0
MOVL C01163 V=800.0 PL=0
MOVL C01164 V=800.0 PL=0
MOVL C01165 V=800.0 PL=0
MOVL C01166 V=800.0 PL=0
MOVL C01167 V=800.0 PL=0
MOVL C01168 V=800.0 PL=0
MOVL C01169 V=800.0 PL=0
MOVL C01170 V=800.0 PL=0
MOVL C01171 V=800.0 PL=0
MOVL C01172 V=800.0 PL=0
MOVL C01173 V=800.0 PL=0
MOVL C01174 V=800.0 PL=0
MOVL C01175 V=800.0 PL=0
MOVL C01176 V=800.0 PL=0
MOVL C01177 V=800.0 PL=0
MOVL C01178 V=800.0 PL=0
MOVL C01179 V=800.0 PL=0
MOVL C01180 V=800.0 PL=0
MOVL C01181 V=800.0 PL=0
MOVL C01182 V=800.0 PL=0
MOVL C01183 V=800.0 PL=0
MOVL C01184 V=800.0 PL=0
MOVL C01185 V=800.0 PL=0
MOVL C01186 V=800.0 PL=0
MOVL C01187 V=800.0 PL=0
MOVL C01188 V=800.0 PL=0
MOVL C01189 V=800.0 PL=0
MOVL C01190 V=800.0 PL=0
MOVL C01191 V=800.0 PL=0
MOVL C01192 V=800.0 PL=0
MOVL C01193 V=800.0 PL=0
MOVL C01194 V=800.0 PL=0
MOVL C01195 V=800.0 PL=0
MOVL C01196 V=800.0 PL=0
MOVL C01197 V=800.0 PL=0
MOVL C01198 V=800.0 PL=0
MOVL C01199 V=800.0 PL=0
MOVL C01200 V=800.0 PL=0
MOVL C01201 V=800.0 PL=0
MOVL C01202 V=800.0 PL=0
MOVL C01203 V=800.0 PL=0
MOVL C01204 V=800.0 PL=0
MOVL C01205 V=800.0 PL=0
MOVL C01206 V=800.0 PL=0
MOVL C01207 V=800.0 PL=0
MOVL C01208 V=800.0 PL=0
MOVL C01209 V=800.0 PL=0
MOVL C01210 V=800.0 PL=0
MOVL C01211 V=800.0 PL=0
MOVL C01212 V=800.0 PL=0
MOVL C01213 V=800.0 PL=0
MOVL C01214 V=800.0 PL=0
MOVL C01215 V=800.0 PL=0
MOVL C01216 V=800.0 PL=0
MOVL C01217 V=800.0 PL=0
MOVL C01218 V=800.0 PL=0
MOVL C01219 V=800.0 PL=0
MOVL C01220 V=800.0 PL=0
MOVL C01221 V=800.0 PL=0
MOVL C01222 V=800.0 PL=0
MOVL C01223 V=800.0 PL=0
MOVL C01224 V=800.0 PL=0
MOVL C01225 V=800.0 PL=0
MOVL C01226 V=800.0 PL=0
MOVL C01227 V=800.0 PL=0
MOVL C01228 V=800.0 PL=0
MOVL C01229 V=800.0 PL=0
MOVL C01230 V=800.0 PL=0
MOVL C01231 V=800.0 PL=0
MOVL C01232 V=800.0 PL=0
MOVL C01233 V=800.0 PL=0
MOVL C01234 V=800.0 PL=0
MOVL C01235 V=800.0 PL=0
MOVL C01236 V=800.0 PL=0
MOVL C01237 V=800.0 PL=0
MOVL C01238 V=800.0 PL=0
MOVL C01239 V=800.0 PL=0
MOVL C01240 V=800.0 PL=0
MOVL C01241 V=800.0 PL=0
MOVL C01242 V=800.0 PL=0
MOVL C01243 V=800.0 PL=0
MOVL C01244 V=800.0 PL=0
MOVL C01245 V=800.0 PL=0
MOVL C01246 V=800.0 PL=0
MOVL C01247 V=800.0 PL=0
MOVL C01248 V=800.0 PL=0
MOVL C01249 V=800.0 PL=0
MOVL C01250 V=800.0 PL=0
MOVL C01251 V=800.0 PL=0
MOVL C01252 V=800.0 PL=0
MOVL C01253 V=800.0 PL=0
MOVL C01254 V=800.0 PL=0
MOVL C01255 V=800.0 PL=0
MOVL C01256 V=800.0 PL=0
MOVL C01257 V=800.0 PL=0
MOVL C01258 V=800.0 PL=0
MOVL C01259 V=800.0 PL=0
MOVL C01260 V=800.0 PL=0
MOVL C01261 V=800.0 PL=0
MOVL C01262 V=800.0 PL=0
MOVL C01263 V=800.0 PL=0
MOVL C01264 V=800.0 PL=0
MOVL C01265 V=800.0 PL=0
MOVL C01266 V=800.0 PL=0
MOVL C01267 V=800.0 PL=0
MOVL C01268 V=800.0 PL=0
MOVL C01269 V=800.0 PL=0
MOVL C01270 V=800.0 PL=0
MOVL C01271 V=800.0 PL=0
MOVL C01272 V=800.0 PL=0
MOVL C01273 V=800.0 PL=0
MOVL C01274 V=800.0 PL=0
MOVL C01275 V=800.0 PL=0
MOVL C01276 V=800.0 PL=0
MOVL C01277 V=800.0 PL=0
MOVL C01278 V=800.0 PL=0
MOVL C01279 V=800.0 PL=0
MOVL C01280 V=800.0 PL=0
MOVL C01281 V=800.0 PL=0
MOVL C01282 V=800.0 PL=0
MOVL C01283 V=800.0 PL=0
MOVL C01284 V=800.0 PL=0
MOVL C01285 V=800.0 PL=0
MOVL C01286 V=800.0 PL=0
MOVL C01287 V=800.0 PL=0
MOVL C01288 V=800.0 PL=0
MOVL C01289 V=800.0 PL=0
MOVL C01290 V=800.0 PL=0
MOVL C01291 V=800.0 PL=0
MOVL C01292 V=800.0 PL=0
MOVL C01293 V=800.0 PL=0
MOVL C01294 V=800.0 PL=0
MOVL C01295 V=800.0 PL=0
MOVL C01296 V=800.0 PL=0
MOVL C01297 V=800.0 PL=0
MOVL C01298 V=800.0 PL=0
MOVL C01299 V=800.0 PL=0
MOVL C01300 V=800.0 PL=0
MOVL C01301 V=800.0 PL=0
MOVL C01302 V=800.0 PL=0
MOVL C01303 V=800.0 PL=0
MOVL C01304 V=800.0 PL=0
MOVL C01305 V=800.0 PL=0
MOVL C01306 V=800.0 PL=0
MOVL C01307 V=800.0 PL=0
MOVL C01308 V=800.0 PL=0
MOVL C01309 V=800.0 PL=0
MOVL C01310 V=800.0 PL=0
MOVL C01311 V=800.0 PL=0
MOVL C01312 V=800.0 PL=0
MOVL C01313 V=800.0 PL=0
MOVL C01314 V=800.0 PL=0
MOVL C01315 V=800.0 PL=0
MOVL C01316 V=800.0 PL=0
MOVL C01317 V=800.0 PL=0
MOVL C01318 V=800.0 PL=0
MOVL C01319 V=800.0 PL=0
MOVL C01320 V=800.0 PL=0
MOVL C01321 V=800.0 PL=0
MOVL C01322 V=800.0 PL=0
MOVL C01323 V=800.0 PL=0
MOVL C01324 V=800.0 PL=0
MOVL C01325 V=800.0 PL=0
MOVL C01326 V=800.0 PL=0
MOVL C01327 V=800.0 PL=0
MOVL C01328 V=800.0 PL=0
MOVL C01329 V=800.0 PL=0
MOVL C01330 V=800.0 PL=0
MOVL C01331 V=800.0 PL=0
MOVL C01332 V=800.0 PL=0
MOVL C01333 V=800.0 PL=0
MOVL C01334 V=800.0 PL=0
MOVL C01335 V=800.0 PL=0
MOVL C01336 V=800.0 PL=0
MOVL C01337 V=800.0 PL=0
MOVL C01338 V=800.0 PL=0
MOVL C01339 V=800.0 PL=0
MOVL C01340 V=800.0 PL=0
MOVL C01341 V=800.0 PL=0
MOVL C01342 V=800.0 PL=0
MOVL C01343 V=800.0 PL=0
MOVL C01344 V=800.0 PL=0
MOVL C01345 V=800.0 PL=0
MOVL C01346 V=800.0 PL=0
MOVL C01347 V=800.0 PL=0
MOVL C01348 V=800.0 PL=0
MOVL C01349 V=800.0 PL=0
MOVL C01350 V=800.0 PL=0
MOVL C01351 V=800.0 PL=0
MOVL C01352 V=800.0 PL=0
MOVL C01353 V=800.0 PL=0
MOVL C01354 V=800.0 PL=0
MOVL C01355 V=800.0 PL=0
MOVL C01356 V=800.0 PL=0
MOVL C01357 V=800.0 PL=0
MOVL C01358 V=800.0 PL=0
MOVL C01359 V=800.0 PL=0
MOVL C01360 V=800.0 PL=0
MOVL C01361 V=800.0 PL=0
MOVL C01362 V=800.0 PL=0
MOVL C01363 V=800.0 PL=0
MOVL C01364 V=800.0 PL=0
MOVL C01365 V=800.0 PL=0
MOVL C01366 V=800.0 PL=0
MOVL C01367 V=800.0 PL=0
MOVL C01368 V=800.0 PL=0
MOVL C01369 V=800.0 PL=0
MOVL C01370 V=800.0 PL=0
MOVL C01371 V=800.0 PL=0
MOVL C01372 V=800.0 PL=0
MOVL C01373 V=800.0 PL=0
MOVL C01374 V=800.0 PL=0
MOVL C01375 V=800.0 PL=0
MOVL C01376 V=800.0 PL=0
MOVL C01377 V=800.0 PL=0
MOVL C01378 V=800.0 PL=0
MOVL C01379 V=800.0 PL=0
MOVL C01380 V=800.0 PL=0
MOVL C01381 V=800.0 PL=0
MOVL C01382 V=800.0 PL=0
MOVL C01383 V=800.0 PL=0
MOVL C01384 V=800.0 PL=0
MOVL C01385 V=800.0 PL=0
MOVL C01386 V=800.0 PL=0
MOVL C01387 V=800.0 PL=0
MOVL C01388 V=800.0 PL=0
MOVL C01389 V=800.0 PL=0
MOVL C01390 V=800.0 PL=0
MOVL C01391 V=800.0 PL=0
MOVL C01392 V=800.0 PL=0
MOVL C01393 V=800.0 PL=0
MOVL C01394 V=800.0 PL=0
MOVL C01395 V=800.0 PL=0
MOVL C01396 V=800.0 PL=0
MOVL C01397 V=800.0 PL=0
MOVL C01398 V=800.0 PL=0
MOVL C01399 V=800.0 PL=0
MOVL C01400 V=800.0 PL=0
MOVL C01401 V=800.0 PL=0
MOVL C01402 V=800.0 PL=0
MOVL C01403 V=800.0 PL=0
MOVL C01404 V=800.0 PL=0
MOVL C01405 V=800.0 PL=0
MOVL C01406 V=800.0 PL=0
MOVL C01407 V=800.0 PL=0
MOVL C01408 V=800.0 PL=0
MOVL C01409 V=800.0 PL=0
MOVL C01410 V=800.0 PL=0
MOVL C01411 V=800.0 PL=0
MOVL C01412 V=800.0 PL=0
MOVL C01413 V=800.0 PL=0
MOVL C01414 V=800.0 PL=0
MOVL C01415 V=800.0 PL=0
MOVL C01416 V=800.0 PL=0
MOVL C01417 V=800.0 PL=0
MOVL C01418 V=800.0 PL=0
MOVL C01419 V=800.0 PL=0
MOVL C01420 V=800.0 PL=0
MOVL C01421 V=800.0 PL=0
MOVL C01422 V=800.0 PL=0
MOVL C01423 V=800.0 PL=0
MOVL C01424 V=800.0 PL=0
MOVL C01425 V=800.0 PL=0
MOVL C01426 V=800.0 PL=0
MOVL C01427 V=800.0 PL=0
MOVL C01428 V=800.0 PL=0
MOVL C01429 V=800.0 PL=0
MOVL C01430 V=800.0 PL=0
MOVL C01431 V=800.0 PL=0
MOVL C01432 V=800.0 PL=0
MOVL C01433 V=800.0 PL=0
MOVL C01434 V=800.0 PL=0
MOVL C01435 V=800.0 PL=0
MOVL C01436 V=800.0 PL=0
MOVL C01437 V=800.0 PL=0
MOVL C01438 V=800.0 PL=0
MOVL C01439 V=800.0 PL=0
MOVL C01440 V=800.0 PL=0
MOVL C01441 V=800.0 PL=0
MOVL C01442 V=800.0 PL=0
MOVL C01443 V=800.0 PL=0
MOVL C01444 V=800.0 PL=0
MOVL C01445 V=800.0 PL=0
MOVL C01446 V=800.0 PL=0
MOVL C01447 V=800.0 PL=0
MOVL C01448 V=800.0 PL=0
MOVL C01449 V=800.0 PL=0
MOVL C01450 V=800.0 PL=0
MOVL C01451 V=800.0 PL=0
MOVL C01452 V=800.0 PL=0
MOVL C01453 V=800.0 PL=0
MOVL C01454 V=800.0 PL=0
MOVL C01455 V=800.0 PL=0
MOVL C01456 V=800.0 PL=0
MOVL C01457 V=800.0 PL=0
MOVL C01458 V=800.0 PL=0
MOVL C01459 V=800.0 PL=0
MOVL C01460 V=800.0 PL=0
MOVL C01461 V=800.0 PL=0
MOVL C01462 V=800.0 PL=0
MOVL C01463 V=800.0 PL=0
MOVL C01464 V=800.0 PL=0
MOVL C01465 V=800.0 PL=0
MOVL C01466 V=800.0 PL=0
MOVL C01467 V=800.0 PL=0
MOVL C01468 V=800.0 PL=0
MOVL C01469 V=800.0 PL=0
MOVL C01470 V=800.0 PL=0
MOVL C01471 V=800.0 PL=0
MOVL C01472 V=800.0 PL=0
MOVL C01473 V=800.0 PL=0
MOVL C01474 V=800.0 PL=0
MOVL C01475 V=800.0 PL=0
MOVL C01476 V=800.0 PL=0
MOVL C01477 V=800.0 PL=0
MOVL C01478 V=800.0 PL=0
MOVL C01479 V=800.0 PL=0
MOVL C01480 V=800.0 PL=0
MOVL C01481 V=800.0 PL=0
MOVL C01482 V=800.0 PL=0
MOVL C01483 V=800.0 PL=0
MOVL C01484 V=800.0 PL=0
MOVL C01485 V=800.0 PL=0
MOVL C01486 V=800.0 PL=0
MOVL C01487 V=800.0 PL=0
MOVL C01488 V=800.0 PL=0
MOVL C01489 V=800.0 PL=0
MOVL C01490 V=800.0 PL=0
MOVL C01491 V=800.0 PL=0
MOVL C01492 V=800.0 PL=0
MOVL C01493 V=800.0 PL=0
MOVL C01494 V=800.0 PL=0
MOVL C01495 V=800.0 PL=0
MOVL C01496 V=800.0 PL=0
MOVL C01497 V=800.0 PL=0
MOVL C01498 V=800.0 PL=0
MOVL C01499 V=800.0 PL=0
MOVL C01500 V=800.0 PL=0
MOVL C01501 V=800.0 PL=0
MOVL C01502 V=800.0 PL=0
MOVL C01503 V=800.0 PL=0
MOVL C01504 V=800.0 PL=0
MOVL C01505 V=800.0 PL=0
MOVL C01506 V=800.0 PL=0
MOVL C01507 V=800.0 PL=0
MOVL C01508 V=800.0 PL=0
MOVL C01509 V=800.0 PL=0
MOVL C01510 V=800.0 PL=0
MOVL C01511 V=800.0 PL=0
MOVL C01512 V=800.0 PL=0
MOVL C01513 V=800.0 PL=0
MOVL C01514 V=800.0 PL=0
MOVL C01515 V=800.0 PL=0
MOVL C01516 V=800.0 PL=0
MOVL C01517 V=800.0 PL=0
MOVL C01518 V=800.0 PL=0
MOVL C01519 V=800.0 PL=0
MOVL C01520 V=800.0 PL=0
MOVL C01521 V=800.0 PL=0
MOVL C01522 V=800.0 PL=0
MOVL C01523 V=800.0 PL=0
MOVL C01524 V=800.0 PL=0
MOVL C01525 V=800.0 PL=0
MOVL C01526 V=800.0 PL=0
MOVL C01527 V=800.0 PL=0
MOVL C01528 V=800.0 PL=0
MOVL C01529 V=800.0 PL=0
MOVL C01530 V=800.0 PL=0
MOVL C01531 V=800.0 PL=0
MOVL C01532 V=800.0 PL=0
MOVL C01533 V=800.0 PL=0
MOVL C01534 V=800.0 PL=0
MOVL C01535 V=800.0 PL=0
MOVL C01536 V=800.0 PL=0
MOVL C01537 V=800.0 PL=0
MOVL C01538 V=800.0 PL=0
MOVL C01539 V=800.0 PL=0
MOVL C01540 V=800.0 PL=0
MOVL C01541 V=800.0 PL=0
MOVL C01542 V=800.0 PL=0
MOVL C01543 V=800.0 PL=0
MOVL C01544 V=800.0 PL=0
MOVL C01545 V=800.0 PL=0
MOVL C01546 V=800.0 PL=0
MOVL C01547 V=800.0 PL=0
MOVL C01548 V=800.0 PL=0
MOVL C01549 V=800.0 PL=0
MOVL C01550 V=800.0 PL=0
MOVL C01551 V=800.0 PL=0
MOVL C01552 V=800.0 PL=0
MOVL C01553 V=800.0 PL=0
MOVL C01554 V=800.0 PL=0
MOVL C01555 V=800.0 PL=0
MOVL C01556 V=800.0 PL=0
MOVL C01557 V=800.0 PL=0
MOVL C01558 V=800.0 PL=0
MOVL C01559 V=800.0 PL=0
MOVL C01560 V=800.0 PL=0
MOVL C01561 V=800.0 PL=0
MOVL C01562 V=800.0 PL=0
MOVL C01563 V=800.0 PL=0
MOVL C01564 V=800.0 PL=0
MOVL C01565 V=800.0 PL=0
MOVL C01566 V=800.0 PL=0
MOVL C01567 V=800.0 PL=0
MOVL C01568 V=800.0 PL=0
MOVL C01569 V=800.0 PL=0
MOVL C01570 V=800.0 PL=0
MOVL C01571 V=800.0 PL=0
MOVL C01572 V=800.0 PL=0
MOVL C01573 V=800.0 PL=0
MOVL C01574 V=800.0 PL=0
MOVL C01575 V=800.0 PL=0
MOVL C01576 V=800.0 PL=0
MOVL C01577 V=800.0 PL=0
MOVL C01578 V=800.0 PL=0
MOVL C01579 V=800.0 PL=0
MOVL C01580 V=800.0 PL=0
MOVL C01581 V=800.0 PL=0
MOVL C01582 V=800.0 PL=0
MOVL C01583 V=800.0 PL=0
MOVL C01584 V=800.0 PL=0
MOVL C01585 V=800.0 PL=0
MOVL C01586 V=800.0 PL=0
MOVL C01587 V=800.0 PL=0
MOVL C01588 V=800.0 PL=0
MOVL C01589 V=800.0 PL=0
MOVL C01590 V=800.0 PL=0
MOVL C01591 V=800.0 PL=0
MOVL C01592 V=800.0 PL=0
MOVL C01593 V=800.0 PL=0
MOVL C01594 V=800.0 PL=0
MOVL C01595 V=800.0 PL=0
MOVL C01596 V=800.0 PL=0
MOVL C01597 V=800.0 PL=0
MOVL C01598 V=800.0 PL=0
MOVL C01599 V=800.0 PL=0
MOVL C01600 V=800.0 PL=0
MOVL C01601 V=800.0 PL=0
MOVL C01602 V=800.0 PL=0
MOVL C01603 V=800.0 PL=0
MOVL C01604 V=800.0 PL=0
MOVL C01605 V=800.0 PL=0
MOVL C01606 V=800.0 PL=0
MOVL C01607 V=800.0 PL=0
MOVL C01608 V=800.0 PL=0
MOVL C01609 V=800.0 PL=0
MOVL C01610 V=800.0 PL=0
MOVL C01611 V=800.0 PL=0
MOVL C01612 V=800.0 PL=0
MOVL C01613 V=800.0 PL=0
MOVL C01614 V=800.0 PL=0
MOVL C01615 V=800.0 PL=0
MOVL C01616 V=800.0 PL=0
MOVL C01617 V=800.0 PL=0
MOVL C01618 V=800.0 PL=0
MOVL C01619 V=800.0 PL=0
MOVL C01620 V=800.0 PL=0
MOVL C01621 V=800.0 PL=0
MOVL C01622 V=800.0 PL=0
MOVL C01623 V=800.0 PL=0
MOVL C01624 V=800.0 PL=0
MOVL C01625 V=800.0 PL=0
MOVL C01626 V=800.0 PL=0
MOVL C01627 V=800.0 PL=0
MOVL C01628 V=800.0 PL=0
MOVL C01629 V=800.0 PL=0
MOVL C01630 V=800.0 PL=0
MOVL C01631 V=800.0 PL=0
MOVL C01632 V=800.0 PL=0
MOVL C01633 V=800.0 PL=0
MOVL C01634 V=800.0 PL=0
MOVL C01635 V=800.0 PL=0
MOVL C01636 V=800.0 PL=0
MOVL C01637 V=800.0 PL=0
MOVL C01638 V=800.0 PL=0
MOVL C01639 V=800.0 PL=0
MOVL C01640 V=800.0 PL=0
MOVL C01641 V=800.0 PL=0
MOVL C01642 V=800.0 PL=0
MOVL C01643 V=800.0 PL=0
MOVL C01644 V=800.0 PL=0
MOVL C01645 V=800.0 PL=0
MOVL C01646 V=800.0 PL=0
MOVL C01647 V=800.0 PL=0
MOVL C01648 V=800.0 PL=0
MOVL C01649 V=800.0 PL=0
MOVL C01650 V=800.0 PL=0
MOVL C01651 V=800.0 PL=0
MOVL C01652 V=800.0 PL=0
MOVL C01653 V=800.0 PL=0
MOVL C01654 V=800.0 PL=0
MOVL C01655 V=800.0 PL=0
MOVL C01656 V=800.0 PL=0
MOVL C01657 V=800.0 PL=0
MOVL C01658 V=800.0 PL=0
MOVL C01659 V=800.0 PL=0
MOVL C01660 V=800.0 PL=0
MOVL C01661 V=800.0 PL=0
MOVL C01662 V=800.0 PL=0
MOVL C01663 V=800.0 PL=0
MOVL C01664 V=800.0 PL=0
MOVL C01665 V=800.0 PL=0
MOVL C01666 V=800.0 PL=0
MOVL C01667 V=800.0 PL=0
MOVL C01668 V=800.0 PL=0
MOVL C01669 V=800.0 PL=0
MOVL C01670 V=800.0 PL=0
MOVL C01671 V=800.0 PL=0
MOVL C01672 V=800.0 PL=0
MOVL C01673 V=800.0 PL=0
MOVL C01674 V=800.0 PL=0
MOVL C01675 V=800.0 PL=0
MOVL C01676 V=800.0 PL=0
MOVL C01677 V=800.0 PL=0
MOVL C01678 V=800.0 PL=0
MOVL C01679 V=800.0 PL=0
MOVL C01680 V=800.0 PL=0
MOVL C01681 V=800.0 PL=0
MOVL C01682 V=800.0 PL=0
MOVL C01683 V=800.0 PL=0
MOVL C01684 V=800.0 PL=0
MOVL C01685 V=800.0 PL=0
MOVL C01686 V=800.0 PL=0
MOVL C01687 V=800.0 PL=0
MOVL C01688 V=800.0 PL=0
MOVL C01689 V=800.0 PL=0
MOVL C01690 V=800.0 PL=0
MOVL C01691 V=800.0 PL=0
MOVL C01692 V=800.0 PL=0
MOVL C01693 V=800.0 PL=0
MOVL C01694 V=800.0 PL=0
MOVL C01695 V=800.0 PL=0
MOVL C01696 V=800.0 PL=0
MOVL C01697 V=800.0 PL=0
MOVL C01698 V=800.0 PL=0
MOVL C01699 V=800.0 PL=0
MOVL C01700 V=800.0 PL=0
MOVL C01701 V=800.0 PL=0
MOVL C01702 V=800.0 PL=0
MOVL C01703 V=800.0 PL=0
MOVL C01704 V=800.0 PL=0
MOVL C01705 V=800.0 PL=0
MOVL C01706 V=800.0 PL=0
MOVL C01707 V=800.0 PL=0
MOVL C01708 V=800.0 PL=0
MOVL C01709 V=800.0 PL=0
MOVL C01710 V=800.0 PL=0
MOVL C01711 V=800.0 PL=0
MOVL C01712 V=800.0 PL=0
MOVL C01713 V=800.0 PL=0
MOVL C01714 V=800.0 PL=0
MOVL C01715 V=800.0 PL=0
MOVL C01716 V=800.0 PL=0
MOVL C01717 V=800.0 PL=0
MOVL C01718 V=800.0 PL=0
MOVL C01719 V=800.0 PL=0
MOVL C01720 V=800.0 PL=0
MOVL C01721 V=800.0 PL=0
MOVL C01722 V=800.0 PL=0
MOVL C01723 V=800.0 PL=0
MOVL C01724 V=800.0 PL=0
MOVL C01725 V=800.0 PL=0
MOVL C01726 V=800.0 PL=0
MOVL C01727 V=800.0 PL=0
MOVL C01728 V=800.0 PL=0
MOVL C01729 V=800.0 PL=0
MOVL C01730 V=800.0 PL=0
MOVL C01731 V=800.0 PL=0
MOVL C01732 V=800.0 PL=0
MOVL C01733 V=800.0 PL=0
MOVL C01734 V=800.0 PL=0
MOVL C01735 V=800.0 PL=0
MOVL C01736 V=800.0 PL=0
MOVL C01737 V=800.0 PL=0
MOVL C01738 V=800.0 PL=0
MOVL C01739 V=800.0 PL=0
MOVL C01740 V=800.0 PL=0
MOVL C01741 V=800.0 PL=0
MOVL C01742 V=800.0 PL=0
MOVL C01743 V=800.0 PL=0
MOVL C01744 V=800.0 PL=0
MOVL C01745 V=800.0 PL=0
MOVL C01746 V=800.0 PL=0
MOVL C01747 V=800.0 PL=0
MOVL C01748 V=800.0 PL=0
MOVL C01749 V=800.0 PL=0
MOVL C01750 V=800.0 PL=0
MOVL C01751 V=800.0 PL=0
MOVL C01752 V=800.0 PL=0
MOVL C01753 V=800.0 PL=0
MOVL C01754 V=800.0 PL=0
MOVL C01755 V=800.0 PL=0
MOVL C01756 V=800.0 PL=0
MOVL C01757 V=800.0 PL=0
MOVL C01758 V=800.0 PL=0
MOVL C01759 V=800.0 PL=0
MOVL C01760 V=800.0 PL=0
MOVL C01761 V=800.0 PL=0
MOVL C01762 V=800.0 PL=0
MOVL C01763 V=800.0 PL=0
MOVL C01764 V=800.0 PL=0
MOVL C01765 V=800.0 PL=0
MOVL C01766 V=800.0 PL=0
MOVL C01767 V=800.0 PL=0
MOVL C01768 V=800.0 PL=0
MOVL C01769 V=800.0 PL=0
MOVL C01770 V=800.0 PL=0
MOVL C01771 V=800.0 PL=0
MOVL C01772 V=800.0 PL=0
MOVL C01773 V=800.0 PL=0
MOVL C01774 V=800.0 PL=0
MOVL C01775 V=800.0 PL=0
MOVL C01776 V=800.0 PL=0
MOVL C01777 V=800.0 PL=0
MOVL C01778 V=800.0 PL=0
MOVL C01779 V=800.0 PL=0
MOVL C01780 V=800.0 PL=0
MOVL C01781 V=800.0 PL=0
MOVL C01782 V=800.0 PL=0
MOVL C01783 V=800.0 PL=0
MOVL C01784 V=800.0 PL=0
MOVL C01785 V=800.0 PL=0
MOVL C01786 V=800.0 PL=0
MOVL C01787 V=800.0 PL=0
MOVL C01788 V=800.0 PL=0
MOVL C01789 V=800.0 PL=0
MOVL C01790 V=800.0 PL=0
MOVL C01791 V=800.0 PL=0
MOVL C01792 V=800.0 PL=0
MOVL C01793 V=800.0 PL=0
MOVL C01794 V=800.0 PL=0
MOVL C01795 V=800.0 PL=0
MOVL C01796 V=800.0 PL=0
MOVL C01797 V=800.0 PL=0
MOVL C01798 V=800.0 PL=0
MOVL C01799 V=800.0 PL=0
MOVL C01800 V=800.0 PL=0
MOVL C01801 V=800.0 PL=0
MOVL C01802 V=800.0 PL=0
MOVL C01803 V=800.0 PL=0
MOVL C01804 V=800.0 PL=0
MOVL C01805 V=800.0 PL=0
MOVL C01806 V=800.0 PL=0
MOVL C01807 V=800.0 PL=0
MOVL C01808 V=800.0 PL=0
MOVL C01809 V=800.0 PL=0
MOVL C01810 V=800.0 PL=0
MOVL C01811 V=800.0 PL=0
MOVL C01812 V=800.0 PL=0
MOVL C01813 V=800.0 PL=0
MOVL C01814 V=800.0 PL=0
MOVL C01815 V=800.0 PL=0
MOVL C01816 V=800.0 PL=0
MOVL C01817 V=800.0 PL=0
MOVL C01818 V=800.0 PL=0
MOVL C01819 V=800.0 PL=0
MOVL C01820 V=800.0 PL=0
MOVL C01821 V=800.0 PL=0
MOVL C01822 V=800.0 PL=0
MOVL C01823 V=800.0 PL=0
MOVL C01824 V=800.0 PL=0
MOVL C01825 V=800.0 PL=0
MOVL C01826 V=800.0 PL=0
MOVL C01827 V=800.0 PL=0
MOVL C01828 V=800.0 PL=0
MOVL C01829 V=800.0 PL=0
MOVL C01830 V=800.0 PL=0
MOVL C01831 V=800.0 PL=0
MOVL C01832 V=800.0 PL=0
MOVL C01833 V=800.0 PL=0
MOVL C01834 V=800.0 PL=0
MOVL C01835 V=800.0 PL=0
MOVL C01836 V=800.0 PL=0
MOVL C01837 V=800.0 PL=0
MOVL C01838 V=800.0 PL=0
MOVL C01839 V=800.0 PL=0
MOVL C01840 V=800.0 PL=0
MOVL C01841 V=800.0 PL=0
MOVL C01842 V=800.0 PL=0
MOVL C01843 V=800.0 PL=0
MOVL C01844 V=800.0 PL=0
MOVL C01845 V=800.0 PL=0
MOVL C01846 V=800.0 PL=0
MOVL C01847 V=800.0 PL=0
MOVL C01848 V=800.0 PL=0
MOVL C01849 V=800.0 PL=0
MOVL C01850 V=800.0 PL=0
MOVL C01851 V=800.0 PL=0
MOVL C01852 V=800.0 PL=0
MOVL C01853 V=800.0 PL=0
MOVL C01854 V=800.0 PL=0
MOVL C01855 V=800.0 PL=0
MOVL C01856 V=800.0 PL=0
MOVL C01857 V=800.0 PL=0
MOVL C01858 V=800.0 PL=0
MOVL C01859 V=800.0 PL=0
MOVL C01860 V=800.0 PL=0
MOVL C01861 V=800.0 PL=0
MOVL C01862 V=800.0 PL=0
MOVL C01863 V=800.0 PL=0
MOVL C01864 V=800.0 PL=0
MOVL C01865 V=800.0 PL=0
MOVL C01866 V=800.0 PL=0
MOVL C01867 V=800.0 PL=0
MOVL C01868 V=800.0 PL=0
MOVL C01869 V=800.0 PL=0
MOVL C01870 V=800.0 PL=0
MOVL C01871 V=800.0 PL=0
MOVL C01872 V=800.0 PL=0
MOVL C01873 V=800.0 PL=0
MOVL C01874 V=800.0 PL=0
MOVL C01875 V=800.0 PL=0
MOVL C01876 V=800.0 PL=0
MOVL C01877 V=800.0 PL=0
MOVL C01878 V=800.0 PL=0
MOVL C01879 V=800.0 PL=0
MOVL C01880 V=800.0 PL=0
MOVL C01881 V=800.0 PL=0
MOVL C01882 V=800.0 PL=0
MOVL C01883 V=800.0 PL=0
MOVL C01884 V=800.0 PL=0
MOVL C01885 V=800.0 PL=0
MOVL C01886 V=800.0 PL=0
MOVL C01887 V=800.0 PL=0
MOVL C01888 V=800.0 PL=0
MOVL C01889 V=800.0 PL=0
MOVL C01890 V=800.0 PL=0
MOVL C01891 V=800.0 PL=0
MOVL C01892 V=800.0 PL=0
MOVL C01893 V=800.0 PL=0
MOVL C01894 V=800.0 PL=0
MOVL C01895 V=800.0 PL=0
MOVL C01896 V=800.0 PL=0
MOVL C01897 V=800.0 PL=0
MOVL C01898 V=800.0 PL=0
MOVL C01899 V=800.0 PL=0
MOVL C01900 V=800.0 PL=0
MOVL C01901 V=800.0 PL=0
MOVL C01902 V=800.0 PL=0
MOVL C01903 V=800.0 PL=0
MOVL C01904 V=800.0 PL=0
MOVL C01905 V=800.0 PL=0
MOVL C01906 V=800.0 PL=0
MOVL C01907 V=800.0 PL=0
MOVL C01908 V=800.0 PL=0
MOVL C01909 V=800.0 PL=0
MOVL C01910 V=800.0 PL=0
MOVL C01911 V=800.0 PL=0
MOVL C01912 V=800.0 PL=0
MOVL C01913 V=800.0 PL=0
MOVL C01914 V=800.0 PL=0
MOVL C01915 V=800.0 PL=0
MOVL C01916 V=800.0 PL=0
MOVL C01917 V=800.0 PL=0
MOVL C01918 V=800.0 PL=0
MOVL C01919 V=800.0 PL=0
MOVL C01920 V=800.0 PL=0
MOVL C01921 V=800.0 PL=0
MOVL C01922 V=800.0 PL=0
MOVL C01923 V=800.0 PL=0
MOVL C01924 V=800.0 PL=0
MOVL C01925 V=800.0 PL=0
MOVL C01926 V=800.0 PL=0
MOVL C01927 V=800.0 PL=0
MOVL C01928 V=800.0 PL=0
MOVL C01929 V=800.0 PL=0
MOVL C01930 V=800.0 PL=0
MOVL C01931 V=800.0 PL=0
MOVL C01932 V=800.0 PL=0
MOVL C01933 V=800.0 PL=0
MOVL C01934 V=800.0 PL=0
MOVL C01935 V=800.0 PL=0
MOVL C01936 V=800.0 PL=0
MOVL C01937 V=800.0 PL=0
MOVL C01938 V=800.0 PL=0
MOVL C01939 V=800.0 PL=0
MOVL C01940 V=800.0 PL=0
MOVL C01941 V=800.0 PL=0
MOVL C01942 V=800.0 PL=0
MOVL C01943 V=800.0 PL=0
MOVL C01944 V=800.0 PL=0
MOVL C01945 V=800.0 PL=0
MOVL C01946 V=800.0 PL=0
MOVL C01947 V=800.0 PL=0
MOVL C01948 V=800.0 PL=0
MOVL C01949 V=800.0 PL=0
MOVL C01950 V=800.0 PL=0
MOVL C01951 V=800.0 PL=0
MOVL C01952 V=800.0 PL=0
MOVL C01953 V=800.0 PL=0
MOVL C01954 V=800.0 PL=0
MOVL C01955 V=800.0 PL=0
MOVL C01956 V=800.0 PL=0
MOVL C01957 V=800.0 PL=0
MOVL C01958 V=800.0 PL=0
MOVL C01959 V=800.0 PL=0
MOVL C01960 V=800.0 PL=0
MOVL C01961 V=800.0 PL=0
MOVL C01962 V=800.0 PL=0
MOVL C01963 V=800.0 PL=0
MOVL C01964 V=800.0 PL=0
MOVL C01965 V=800.0 PL=0
MOVL C01966 V=800.0 PL=0
MOVL C01967 V=800.0 PL=0
MOVL C01968 V=800.0 PL=0
MOVL C01969 V=800.0 PL=0
MOVL C01970 V=800.0 PL=0
MOVL C01971 V=800.0 PL=0
MOVL C01972 V=800.0 PL=0
MOVL C01973 V=800.0 PL=0
MOVL C01974 V=800.0 PL=0
MOVL C01975 V=800.0 PL=0
MOVL C01976 V=800.0 PL=0
MOVL C01977 V=800.0 PL=0
MOVL C01978 V=800.0 PL=0
MOVL C01979 V=800.0 PL=0
MOVL C01980 V=800.0 PL=0
MOVL C01981 V=800.0 PL=0
MOVL C01982 V=800.0 PL=0
MOVL C01983 V=800.0 PL=0
MOVL C01984 V=800.0 PL=0
MOVL C01985 V=800.0 PL=0
MOVL C01986 V=800.0 PL=0
MOVL C01987 V=800.0 PL=0
MOVL C01988 V=800.0 PL=0
MOVL C01989 V=800.0 PL=0
MOVL C01990 V=800.0 PL=0
MOVL C01991 V=800.0 PL=0
MOVL C01992 V=800.0 PL=0
MOVL C01993 V=800.0 PL=0
MOVL C01994 V=800.0 PL=0
MOVL C01995 V=800.0 PL=0
MOVL C01996 V=800.0 PL=0
MOVL C01997 V=800.0 PL=0
MOVL C01998 V=800.0 PL=0
MOVL C01999 V=800.0 PL=0
MOVL C02000 V=800.0 PL=0
MOVL C02001 V=800.0 PL=0
MOVL C02002 V=800.0 PL=0
MOVL C02003 V=800.0 PL=0
MOVL C02004 V=800.0 PL=0
MOVL C02005 V=800.0 PL=0
MOVL C02006 V=800.0 PL=0
MOVL C02007 V=800.0 PL=0
MOVL C02008 V=800.0 PL=0
MOVL C02009 V=800.0 PL=0
MOVL C02010 V=800.0 PL=0
MOVL C02011 V=800.0 PL=0
MOVL C02012 V=800.0 PL=0
MOVL C02013 V=800.0 PL=0
MOVL C02014 V=800.0 PL=0
MOVL C02015 V=800.0 PL=0
MOVL C02016 V=800.0 PL=0
MOVL C02017 V=800.0 PL=0
MOVL C02018 V=800.0 PL=0
MOVL C02019 V=800.0 PL=0
MOVL C02020 V=800.0 PL=0
MOVL C02021 V=800.0 PL=0
MOVL C02022 V=800.0 PL=0
MOVL C02023 V=800.0 PL=0
MOVL C02024 V=800.0 PL=0
MOVL C02025 V=800.0 PL=0
MOVL C02026 V=800.0 PL=0
MOVL C02027 V=800.0 PL=0
MOVL C02028 V=800.0 PL=0
MOVL C02029 V=800.0 PL=0
MOVL C02030 V=800.0 PL=0
MOVL C02031 V=800.0 PL=0
MOVL C02032 V=800.0 PL=0
MOVL C02033 V=800.0 PL=0
MOVL C02034 V=800.0 PL=0
MOVL C02035 V=800.0 PL=0
MOVL C02036 V=800.0 PL=0
MOVL C02037 V=800.0 PL=0
MOVL C02038 V=800.0 PL=0
MOVL C02039 V=800.0 PL=0
MOVL C02040 V=800.0 PL=0
MOVL C02041 V=800.0 PL=0
MOVL C02042 V=800.0 PL=0
MOVL C02043 V=800.0 PL=0
MOVL C02044 V=800.0 PL=0
MOVL C02045 V=800.0 PL=0
MOVL C02046 V=800.0 PL=0
MOVL C02047 V=800.0 PL=0
